(* IEC 61131-3 sources: std_i2980_v2.06_cp053/Source/IMM/ieccontrol/ServiceNet (part 3) *)

         aScan(Execute := FALSE);
      END_IF;
      // next symbol ...
      aScan(Execute := TRUE);
   UNTIL ((NOT aScan.Done) OR (iCntTimeOut = 0))
   END_REPEAT;
ELSE
   // execute false ... clear var outputs and local variables
   bExecuteOld := Execute;
   IF (mHdlNumDataTable <> EMPTY) THEN
      s := KMEM_HashMapL_Delete(mHdlNumDataTable);
      mHdlNumDataTable := EMPTY;
   END_IF;

   iState := 0;
   Error := FALSE;
   sErrMsg := '';
   sParent := '';
   iKeyPosStackIdx := 0;
   ObjRcvCnt := 0;
   iCntStartToken := 0;
   iArrayRecCnt := 0;
   ElapsedTimeSinceLastObj := T#0ms;
END_IF;

@END_Body

@@@BEG_Comment@@@
@TL(39)
@h    ! WARNING !
@h    The Kemro K2 system (including software) only meets category B according to EN 954-1,
@h    thus it is not intended for usage in safety-relevant control applications in the field
@h    of personal safety (e.g. emergency stop).
@h    To implement potentially necessary safety-relevant control tasks, always use additional
@h    external safety devices that are intended for the particular purpose, and meet the necessary
@h    functional safety.
@h    For further information see EN 954-1 (EN ISO 13849-1) and/or the K2-x00 user manual, chapter
@h    "CE conformity, directives and standards".

Algorithm for parsing data stream sent by ServiceNet Server
data presentation: JSON (see http://www.json.org/)

syntax restrictions:
  -> no syntax evaluation of data type "array", tokens within an array are skipped
  -> recursion level for data type "object" is 255 maximum

semantic actions implemented for key - value pairs with values of type "number",
  "true", "false" and "object"

output of parsed data is stored in a hashtable.

objects defined recursive are represented "flat" in same hashtable by adding the parent key
separated by a "." as a prefix to the object key.

the hashtable and it's content is deleted only when reseting input "Execute",
so received data is available in hashtable even if it has not been sent in the
latest message.

data types in hashtable:
-> int numbers, true, false: 4 bytes signed integer (DINT)
-> numbers containing '.' or 'e'/'E': 4 byte float (REAL)

functions available to get a DINT or a REAL value from hashtable.

additionally the parser measures the time since last complete object has
been received for easy timeout detection in calling block.

see documentation for a detailed description.
@@@END_Comment@@@

@BEG_Body
@TL(8)
(**************************************** WARNING ********************************************
 *** The KEBA Kemro K2 System including software is not intended for safety control tasks! ***
 ***                       For further information see Comment tab!                        ***
 *********************************************************************************************)

s := KMEM_HashMapGet(mHdlNumDataTable, Key, Value);
fGetNumValue := s = KMEM_Status_OK;

@END_Body

@@@BEG_Comment@@@
@TL(14)
@h    ! WARNING !
@h    The Kemro K2 system (including software) only meets category B according to EN 954-1,
@h    thus it is not intended for usage in safety-relevant control applications in the field
@h    of personal safety (e.g. emergency stop).
@h    To implement potentially necessary safety-relevant control tasks, always use additional
@h    external safety devices that are intended for the particular purpose, and meet the necessary
@h    functional safety.
@h    For further information see EN 954-1 (EN ISO 13849-1) and/or the K2-x00 user manual, chapter
@h    "CE conformity, directives and standards".

PRIVATE. Not intended to be called from outside this block.

returns the value of a numeric data item stored in hashtable mapped by a certain key
TRUE if found, FALSE in case of an error
@@@END_Comment@@@

@BEG_Body
@TL(15)
(**************************************** WARNING ********************************************
 *** The KEBA Kemro K2 System including software is not intended for safety control tasks! ***
 ***                       For further information see Comment tab!                        ***
 *********************************************************************************************)

bFound := fGetNumValue(Key, tmpValue);
IF ((bFound) AND (tmpValue.dataType = nDTInt)) THEN
   bFound := TRUE;
   ioValue := DWORD_TO_DINT(tmpValue.data);
ELSE
   bFound := FALSE;
END_IF;

fGetDINTValue := bFound;

@END_Body

@@@BEG_Comment@@@
@TL(14)
@h    ! WARNING !
@h    The Kemro K2 system (including software) only meets category B according to EN 954-1,
@h    thus it is not intended for usage in safety-relevant control applications in the field
@h    of personal safety (e.g. emergency stop).
@h    To implement potentially necessary safety-relevant control tasks, always use additional
@h    external safety devices that are intended for the particular purpose, and meet the necessary
@h    functional safety.
@h    For further information see EN 954-1 (EN ISO 13849-1) and/or the K2-x00 user manual, chapter
@h    "CE conformity, directives and standards".

PRIVATE. Not intended to be called from outside this block.

returns the value of a DINT data item stored in hashtable mapped by a certain key
TRUE if found, FALSE in case of an error
@@@END_Comment@@@

@BEG_Body
@TL(18)
(**************************************** WARNING ********************************************
 *** The KEBA Kemro K2 System including software is not intended for safety control tasks! ***
 ***                       For further information see Comment tab!                        ***
 *********************************************************************************************)

IF ((Execute = TRUE) AND (bExecOld = FALSE)) THEN
    // raising edge .. immediate, otherwise if new object recieved since last call
   iCntOld := aParse.ObjRcvCnt - 1;
   bFound := FALSE;
END_IF;

IF (aParse.ObjRcvCnt <> iCntOld) THEN
   bFound := fGetDINTValue(Key, iValue);
   iCntOld := aParse.ObjRcvCnt;
END_IF;

bExecOld := Execute;

@END_Body

@@@BEG_Comment@@@
@TL(15)
@h    ! WARNING !
@h    The Kemro K2 system (including software) only meets category B according to EN 954-1,
@h    thus it is not intended for usage in safety-relevant control applications in the field
@h    of personal safety (e.g. emergency stop).
@h    To implement potentially necessary safety-relevant control tasks, always use additional
@h    external safety devices that are intended for the particular purpose, and meet the necessary
@h    functional safety.
@h    For further information see EN 954-1 (EN ISO 13849-1) and/or the K2-x00 user manual, chapter
@h    "CE conformity, directives and standards".

PRIVATE. Not intended to be called from outside this block.

returns the value of a DINT data item stored in hashtable mapped by a certain key
if not found on raising edge of Execute,
the algorithm will try to find the value each time a new object has been parsed
@@@END_Comment@@@

@BEG_Body
@TL(11)
(**************************************** WARNING ********************************************
 *** The KEBA Kemro K2 System including software is not intended for safety control tasks! ***
 ***                       For further information see Comment tab!                        ***
 *********************************************************************************************)

bFound := fGetNumValue(Key, tmpValue);
IF (bFound) THEN
   bFound := CONVERT_DWORD_TO_REAL(tmpValue.data, rValue);
END_IF;
fGetRealValue := bFound;

@END_Body

@@@BEG_Comment@@@
@TL(14)
@h    ! WARNING !
@h    The Kemro K2 system (including software) only meets category B according to EN 954-1,
@h    thus it is not intended for usage in safety-relevant control applications in the field
@h    of personal safety (e.g. emergency stop).
@h    To implement potentially necessary safety-relevant control tasks, always use additional
@h    external safety devices that are intended for the particular purpose, and meet the necessary
@h    functional safety.
@h    For further information see EN 954-1 (EN ISO 13849-1) and/or the K2-x00 user manual, chapter
@h    "CE conformity, directives and standards".

PRIVATE. Not intended to be called from outside this block.

returns the value of a REAL data item stored in hashtable mapped by a certain key
TRUE if found, FALSE in case of an error
@@@END_Comment@@@

@BEG_Body
@TL(18)
(**************************************** WARNING ********************************************
 *** The KEBA Kemro K2 System including software is not intended for safety control tasks! ***
 ***                       For further information see Comment tab!                        ***
 *********************************************************************************************)

IF ((Execute = TRUE) AND (bExecOld = FALSE)) THEN
   // raising edge .. immediate, otherwise if new object recieved since last call
   iCntOld := aParse.ObjRcvCnt - 1;
   bFound := FALSE;
END_IF;

IF (aParse.ObjRcvCnt <> iCntOld) THEN
   bFound := fGetRealValue(Key, rValue);
   iCntOld := aParse.ObjRcvCnt;
END_IF;

bExecOld := Execute;

@END_Body

@@@BEG_Comment@@@
@TL(13)
@h    ! WARNING !
@h    The Kemro K2 system (including software) only meets category B according to EN 954-1,
@h    thus it is not intended for usage in safety-relevant control applications in the field
@h    of personal safety (e.g. emergency stop).
@h    To implement potentially necessary safety-relevant control tasks, always use additional
@h    external safety devices that are intended for the particular purpose, and meet the necessary
@h    functional safety.
@h    For further information see EN 954-1 (EN ISO 13849-1) and/or the K2-x00 user manual, chapter
@h    "CE conformity, directives and standards".

returns the value of a REAL data item stored in hashtable mapped by a certain key
if not found on raising edge of Execute,
the algorithm will try to find the value each time a new object has been parsed
@@@END_Comment@@@
@END_Body

@END_Contents

(* ---- ABRemoteMaintenance.pu ---- *)
(*
@h    ! WARNING !
@h    The Kemro K2 system (including software) only meets category B according to EN 954-1,
@h    thus it is not intended for usage in safety-relevant control applications in the field
@h    of personal safety (e.g. emergency stop).
@h    To implement potentially necessary safety-relevant control tasks, always use additional
@h    external safety devices that are intended for the particular purpose, and meet the necessary
@h    functional safety.
@h    For further information see EN 954-1 (EN ISO 13849-1) and/or the K2-x00 user manual, chapter
@h    "CE conformity, directives and standards".

This AB controls the logic for connecting ServiceNet via the ServiceNet embedded functionality
via the Remote Maintenance software unit.
*)

IMPORT_OVER_LISTFILE
 KSYS_BPAPI_VAR_READ
, KSYS_BPAPI_VAR_WRITE
, GET_RUNTIME
, KCAT_GetValue
, KCAT_GetHandle
, STOP_PROCESS_ALGORITHM
, START_PROCESS_ALGORITHM
, TOLOWER
, cKSYS_BPApiStateOk
, tsNetworkCfg
, tsTraceLevel
, tsSiteManagerStatus
, TON
, KSYS_BPApiState
, KCAT_HandleData
, KCAT_Status

END_IMPORT

ALGORITHM_BLOCK ABRemoteMaintenance #DUMMY_EDIT_BLOCK

SYSTEM_VAR
 sv_SNNetworkConfig : tsNetworkCfg (* network config to use when connecting to servicenet *);
 sv_iCpuId : LINT;
 sv_TraceLevel : tsTraceLevel;
 sv_bRemoteMaintAvailable : BOOL (* True, if the remote maintenance service is available (Linux only) *);
 sv_bRemoteMaintActivate : BOOL (* Set to true, to activate the remote maintenance *);
 sv_bRemoteMaintActivated : BOOL (* True, if the remote maintenance is activated *);
 sv_sSiteManagerSetServer : STRING(255) (* The SiteManager server name to connect *);
 sv_sSiteManagerSetName : STRING(255) (* The SiteManager domain to connect *);
 sv_iRemoteMaintState : UDINT (* State of the remote maintenance service (1=active) *);
 sv_SiteManager : tsSiteManagerStatus (* Secomea SiteManager structure *);
 sv_bInitStart : BOOL;
END_VAR

SYSTEM_OBJECT
 TaskVis : TASK;
 TaskVisLow : TASK;
END_OBJECT

VAR
 fbTimer : TON;
 mbInit : BOOL;
END_VAR

ALGORITHM aReadSiteManagerStatus

VAR
 SysState : KSYS_BPApiState;
 sTmp : STRING(255);
 dummy : DINT;
END_VAR
#BEGIN_EDIT_BLOCK
(**************************************** WARNING ********************************************
 *** The KEBA Kemro K2 System including software is not intended for safety control tasks! ***
 ***                       For further information see Comment tab!                        ***
 *********************************************************************************************)

SysState := KSYS_BPAPI_VAR_READ('SYS.SERVICES.RemoteMaintenance.Secomea.Sitemanager.status', sTmp);
IF(SysState = cKSYS_BPApiStateOk) THEN
   sv_SiteManager.sState := sTmp;
ELSIF(sv_TraceLevel.bApplication) THEN
   dummy := Print("Remote maintenance: Site manager status cant be read");
END_IF;

SysState := KSYS_BPAPI_VAR_TXTREAD('SYS.SERVICES.RemoteMaintenance.Secomea.Sitemanager.color', sTmp);
IF(SysState = cKSYS_BPApiStateOk) THEN
   sTmp := TOLOWER(sTmp);
   sv_SiteManager.sColor := sTmp;

   // currently the modem status can only be determined with the status string returned
   IF(sTmp = 'red') THEN
      sv_SiteManager.iState := 1;
   ELSIF(sTmp = 'yellow') THEN
      sv_SiteManager.iState := 2;
   ELSIF(sTmp = 'green') THEN
      sv_SiteManager.iState := 3;
   ELSIF(sTmp = 'blue') THEN
      sv_SiteManager.iState := 4;
   ELSE
      sv_SiteManager.iState := 0;
   END_IF;

   sv_SiteManager.bConnected := (sv_SiteManager.iState = 4);

ELSIF(sv_TraceLevel.bApplication) THEN
   dummy := Print("Remote maintenance: Site manager color cant be read");
   sv_SiteManager.bConnected := FALSE;
END_IF;

;#END_EDIT_BLOCK END_ALGORITHM

ALGORITHM aReadSiteManagerServer

VAR
 SysState : KSYS_BPApiState;
 sTmp : STRING(255);
 dummy : DINT;
END_VAR
#BEGIN_EDIT_BLOCK
(**************************************** WARNING ********************************************
 *** The KEBA Kemro K2 System including software is not intended for safety control tasks! ***
 ***                       For further information see Comment tab!                        ***
 *********************************************************************************************)

SysState := KSYS_BPAPI_VAR_TXTREAD('SYS.CFG.Secomea.Sitemanager.Server', sTmp);
IF(SysState = cKSYS_BPApiStateOk) THEN
   sv_SiteManager.sServer := sTmp;
ELSIF(sv_TraceLevel.bApplication) THEN
   dummy := Print("Remote maintenance: Site manager server cant be read");
END_IF;

SysState := KSYS_BPAPI_VAR_TXTREAD('SYS.CFG.Secomea.Sitemanager.Name', sTmp);
IF(SysState = cKSYS_BPApiStateOk) THEN
   sv_SiteManager.sName := sTmp;
ELSIF(sv_TraceLevel.bApplication) THEN
   dummy := Print("Remote maintenance: Site manager name cant be read");
END_IF;

SysState := KSYS_BPAPI_VAR_TXTREAD('SYS.CFG.Secomea.Sitemanager.Domain', sTmp);
IF(SysState = cKSYS_BPApiStateOk) THEN
   sv_SiteManager.sDomain := sTmp;
ELSIF(sv_TraceLevel.bApplication) THEN
   dummy := Print("Remote maintenance: Site manager domain cant be read");
END_IF;

;#END_EDIT_BLOCK END_ALGORITHM

PROCESS_ALGORITHM paRun ON TaskVisLow

VAR
 iRemoteMaintState : UDINT;
 SysState : KSYS_BPApiState;
 dummy : DINT;
 t : TIME;
 iTime : DINT;
 iStep : DINT;
END_VAR
#BEGIN_EDIT_BLOCK
(**************************************** WARNING ********************************************
 *** The KEBA Kemro K2 System including software is not intended for safety control tasks! ***
 ***                       For further information see Comment tab!                        ***
 *********************************************************************************************)

t := GET_RUNTIME();

IF iStep = 0 THEN
   fbTimer(IN := FALSE, PT := t#500ms);
   iStep := 1;
END_IF;

IF iStep = 1 THEN
   fbTimer(IN := TRUE);
   IF(fbTimer.Q) THEN
      iStep := 5;
   END_IF;
END_IF;

IF iStep = 5 THEN
   SysState := KSYS_BPAPI_VAR_READ('SYS.SERVICES.RemoteMaintenance.Secomea.state', iRemoteMaintState);
   IF(SysState <> cKSYS_BPApiStateOk) THEN
      IF(sv_TraceLevel.bApplication) THEN
         dummy := Print("Remote maintenance service not found, KSYS_BPApiState %x", SysState);
      END_IF;
      sv_bRemoteMaintAvailable := FALSE;
      STOP_PROCESS_ALGORITHM(paRun);
      RETURN;
   END_IF;

   IF iRemoteMaintState <> 0 THEN
      // continuously poll for the connection status if the state is active
      // IEC does not have a method for post-updating a BPAPI variable
      aReadSiteManagerStatus();
   ELSIF sv_iRemoteMaintState <> 0 THEN
      // reset the connection status
      IF(sv_SiteManager.sState <> 'disabled') THEN
         sv_SiteManager.sState := 'disabled';
      END_IF;
      IF(sv_SiteManager.sColor <> '') THEN
         sv_SiteManager.sColor := '';
         sv_SiteManager.iState := 0;
      END_IF;
      sv_SiteManager.bConnected := FALSE;
   END_IF;

   sv_iRemoteMaintState := iRemoteMaintState;

   fbTimer(IN := FALSE);
   iStep := 0;
END_IF;

t := GET_RUNTIME() - t;
iTime := LINT_TO_DINT(TIME_TO_LINT(t) / 1000);
IF(iTime >= 10 AND sv_TraceLevel.bApplication) THEN
   dummy := Print("Remote maintenance: Runtime of ABRemoteMaintenance.paRun %d ms", iTime);
END_IF;

;#END_EDIT_BLOCK END_ALGORITHM

POSTUPDATE_ALGORITHM pUpdateServer ON TaskVis WITH sv_sSiteManagerSetServer

VAR
 dummy : DINT;
 SysState : KSYS_BPApiState;
END_VAR
#BEGIN_EDIT_BLOCK
(**************************************** WARNING ********************************************
 *** The KEBA Kemro K2 System including software is not intended for safety control tasks! ***
 ***                       For further information see Comment tab!                        ***
 *********************************************************************************************)

IF (NOT mbInit) THEN
   RETURN;
END_IF;

IF(sv_bRemoteMaintAvailable) THEN
   SysState := KSYS_BPAPI_VAR_WRITE('SYS.CFG.Secomea.Sitemanager.Server', sv_sSiteManagerSetServer);
   IF(SysState <> cKSYS_BPApiStateOk) THEN
      dummy := Print("Remote maintenance: Could not set site manager server, KSYS_BPApiState %x", SysState);
      sv_bRemoteMaintActivate := FALSE;
   END_IF;

   aReadSiteManagerServer();

END_IF;

;#END_EDIT_BLOCK END_ALGORITHM

POSTUPDATE_ALGORITHM pUpdateName ON TaskVis WITH sv_sSiteManagerSetName

VAR
 dummy : DINT;
 SysState : KSYS_BPApiState;
 sTmp : STRING(255);
END_VAR
#BEGIN_EDIT_BLOCK
(**************************************** WARNING ********************************************
 *** The KEBA Kemro K2 System including software is not intended for safety control tasks! ***
 ***                       For further information see Comment tab!                        ***
 *********************************************************************************************)

IF (NOT mbInit) THEN
   RETURN;
END_IF;

IF(sv_bRemoteMaintAvailable) THEN

   sTmp := CONCAT(LINT_TO_STRING(sv_iCpuId), '_', sv_sSiteManagerSetName);
   SysState := KSYS_BPAPI_VAR_WRITE('SYS.CFG.Secomea.Sitemanager.Name', sTmp);
   IF(SysState <> cKSYS_BPApiStateOk) THEN
      dummy := Print("Remote maintenance: Could not set site manager name, KSYS_BPApiState %x", SysState);
      sv_bRemoteMaintActivate := FALSE;
   END_IF;

   aReadSiteManagerServer();

END_IF;

;#END_EDIT_BLOCK END_ALGORITHM

POSTUPDATE_ALGORITHM pInit ON TaskVis WITH sv_bInitStart

VAR
 dummy : DINT;
 SysState : KSYS_BPApiState;
 iRemoteMaintState : UDINT;
 bRemoteMaintActive : BOOL;
 sSecomeaDomain : STRING(255);
 iTemp : DINT;
 b : BOOL;
 bLinux : BOOL;
 HandleData : KCAT_HandleData;
 Status : KCAT_Status;
 sTemp : STRING(255);
 sFind : STRING(32);
END_VAR
#BEGIN_EDIT_BLOCK
(**************************************** WARNING ********************************************
 *** The KEBA Kemro K2 System including software is not intended for safety control tasks! ***
 ***                       For further information see Comment tab!                        ***
 *********************************************************************************************)

HandleData := KCAT_GetHandle('UOS.System');
IF HandleData.Status = KCAT_Status_OK THEN
   Status := KCAT_GetValue(Handle := HandleData.Handle, Buffer := sTemp);
   IF (sTemp = 'Linux') THEN
      bLinux := TRUE;
   END_IF;
END_IF;

IF(NOT bLinux) THEN
   // do not create the nodes on VxWorks - this info does not exist
   // stop and return
   sv_bRemoteMaintAvailable := FALSE;
   STOP_PROCESS_ALGORITHM(paRun);
   RETURN;
END_IF;

// check if RemoteMaintenance software unit is present
SysState := KSYS_BPAPI_VAR_READ('SYS.SERVICES.RemoteMaintenance.Secomea.state', iRemoteMaintState);
IF(SysState <> cKSYS_BPApiStateOk) THEN
   IF(sv_TraceLevel.bApplication) THEN
      dummy := Print("Remote maintenance: service/state not found - stopping, KSYS_BPApiState %x", SysState);
   END_IF;
   // stop and return
   sv_bRemoteMaintAvailable := FALSE;
   STOP_PROCESS_ALGORITHM(paRun);
   RETURN;
END_IF;

// Domain must also be configured
SysState := KSYS_BPAPI_VAR_READ('SYS.CFG.Secomea.Sitemanager.Domain', sSecomeaDomain);
IF(SysState <> cKSYS_BPApiStateOk) THEN
   IF(sv_TraceLevel.bApplication) THEN
      dummy := Print("Remote maintenance: service/domain not found - stopping, KSYS_BPApiState %x", SysState);
   END_IF;
   // stop and return
   sv_bRemoteMaintAvailable := FALSE;
   STOP_PROCESS_ALGORITHM(paRun);
   RETURN;
END_IF;

SysState := KSYS_BPAPI_VAR_READ('SYS.SERVICES.RemoteMaintenance.Secomea.activated', bRemoteMaintActive);
IF(SysState <> cKSYS_BPApiStateOk) THEN
   dummy := Print("Remote maintenance: activated flag not found - setting ignored, KSYS_BPApiState %x", SysState);
   RETURN;
END_IF;
sv_bRemoteMaintActivated := bRemoteMaintActive;
b := WRITE_SV_DIRECT(sv_bRemoteMaintActivate, bRemoteMaintActive);

aReadSiteManagerStatus();
aReadSiteManagerServer();

// initialize the setter variables
sv_sSiteManagerSetServer := sv_SiteManager.sServer;

// prepend <CPUID>_ to the display string
sFind := CONCAT(LINT_TO_STRING(sv_iCpuId), '_');
iTemp := FIND(sv_SiteManager.sName, sFind);

IF (iTemp = 1) THEN
   sv_sSiteManagerSetName := RIGHT(sv_SiteManager.sName, LEN(sv_SiteManager.sName)- LEN(sFind));
ELSE
   sv_sSiteManagerSetName := sv_SiteManager.sName;
END_IF;

sv_iRemoteMaintState := iRemoteMaintState;

// disable ServiceNet IP-switching per default
sv_SNNetworkConfig.sIP := '';

// RemoteMaintenance is available start polling for status changes
sv_bRemoteMaintAvailable := TRUE;
START_PROCESS_ALGORITHM(paRun);

mbInit := TRUE;

;#END_EDIT_BLOCK END_ALGORITHM

POSTUPDATE_ALGORITHM pActivate ON TaskVis WITH sv_bRemoteMaintActivate

VAR
 bRemoteMaintActive : BOOL;
 SysState : KSYS_BPApiState;
 dummy : DINT;
END_VAR
#BEGIN_EDIT_BLOCK
(**************************************** WARNING ********************************************
 *** The KEBA Kemro K2 System including software is not intended for safety control tasks! ***
 ***                       For further information see Comment tab!                        ***
 *********************************************************************************************)

// read the current activation status
SysState := KSYS_BPAPI_VAR_READ('SYS.SERVICES.RemoteMaintenance.Secomea.activated', bRemoteMaintActive);
IF(SysState <> cKSYS_BPApiStateOk) THEN
   dummy := Print("Remote maintenance: activated flag not found - setting ignored, KSYS_BPApiState %x", SysState);
   RETURN;
END_IF;

IF(sv_bRemoteMaintActivate = bRemoteMaintActive) THEN
   sv_bRemoteMaintActivated := bRemoteMaintActive;
   RETURN;
END_IF;

// activate service
SysState := KSYS_BPAPI_VAR_WRITE('SYS.SERVICES.RemoteMaintenance.Secomea.activated', sv_bRemoteMaintActivate);
IF(SysState <> cKSYS_BPApiStateOk) THEN
   dummy := Print("Remote maintenance: activated flag not found - could not set, KSYS_BPApiState %x", SysState);
   sv_bRemoteMaintActivate := FALSE;
   RETURN;
END_IF;

sv_bRemoteMaintActivated := sv_bRemoteMaintActivate;

;#END_EDIT_BLOCK END_ALGORITHM

END_ALGORITHM_BLOCK

#END_OF_IEC_PART

@Puma @IecEditor 6 180 @Pou 25
@@@BEG_Comment@@@
@h    ! WARNING !
@h    The Kemro K2 system (including software) only meets category B according to EN 954-1,
@h    thus it is not intended for usage in safety-relevant control applications in the field
@h    of personal safety (e.g. emergency stop).
@h    To implement potentially necessary safety-relevant control tasks, always use additional
@h    external safety devices that are intended for the particular purpose, and meet the necessary
@h    functional safety.
@h    For further information see EN 954-1 (EN ISO 13849-1) and/or the K2-x00 user manual, chapter
@h    "CE conformity, directives and standards".

This AB controls the logic for connecting ServiceNet via the ServiceNet embedded functionality
via the Remote Maintenance software unit.
@@@END_Comment@@@

@BEG_Contents

@BEG_Func
@RT(17)FuncTreeContainer
8
@Var @RT(19)KSYS_BPAPI_VAR_READ @RT(0) @T @T @DERIVED 0 @F @RT(22)KEBA_STANDARD_FUNCTION @F
@T
@BEG_Attrib
0 @RT(0) @RT(0)
@END_Attrib
1 1 @F @F @F @F

@Var @RT(20)KSYS_BPAPI_VAR_WRITE @RT(0) @T @T @DERIVED 0 @F @RT(22)KEBA_STANDARD_FUNCTION @F
@T
@BEG_Attrib
0 @RT(0) @RT(0)
@END_Attrib
1 1 @F @F @F @F

@Var @RT(11)GET_RUNTIME @RT(0) @T @T @DERIVED 0 @F @RT(22)KEBA_STANDARD_FUNCTION @F
@T
@BEG_Attrib
0 @RT(0) @RT(0)
@END_Attrib
1 1 @F @F @F @F

@Var @RT(13)KCAT_GetValue @RT(0) @T @T @DERIVED 0 @F @RT(22)KEBA_STANDARD_FUNCTION @F
@T
@BEG_Attrib
0 @RT(0) @RT(0)
@END_Attrib
1 1 @F @F @F @F

@Var @RT(14)KCAT_GetHandle @RT(0) @T @T @DERIVED 0 @F @RT(22)KEBA_STANDARD_FUNCTION @F
@T
@BEG_Attrib
0 @RT(0) @RT(0)
@END_Attrib
1 1 @F @F @F @F

@Var @RT(22)STOP_PROCESS_ALGORITHM @RT(0) @T @T @DERIVED 0 @F @RT(23)KEBA_STANDARD_PROCEDURE @F
@T
@BEG_Attrib
0 @RT(0) @RT(0)
@END_Attrib
1 1 @F @F @F @F

@Var @RT(23)START_PROCESS_ALGORITHM @RT(0) @T @T @DERIVED 0 @F @RT(23)KEBA_STANDARD_PROCEDURE @F
@T
@BEG_Attrib
0 @RT(0) @RT(0)
@END_Attrib
1 1 @F @F @F @F

@Var @RT(7)TOLOWER @RT(0) @T @T @DERIVED 0 @F @RT(22)KEBA_STANDARD_FUNCTION @F
@T
@BEG_Attrib
0 @RT(0) @RT(0)
@END_Attrib
1 1 @F @F @F @F

@END_Func

@BEG_Const
@RT(18)ConstTreeContainer
1
@Var @RT(18)cKSYS_BPApiStateOk @RT(0) @T @F @DT @RT(5)DWORD @RT(0) @T @T @BASIC 0 @F
@F @F
@T
@BEG_Attrib
0 @RT(4)16#0 @RT(0)
@END_Attrib
1 1 @F @F @F @F

@END_Const

@BEG_Export

@BEG_Kind
@ALGORITHM_BLOCK @RT(19)ABRemoteMaintenance @STRUCTURED_TEXT
@RT(0) @RT(0) @RT(0)
@END_Kind

@BEG_Dcl
@RT(16)DclTreeContainer
15
@Var @RT(7)TaskVis @RT(0) @T @T @RENAMED 0 @T @T @DT @RT(4)TASK @RT(0) @T @T @BASIC 0 @F
@F @F
@T
@BEG_Attrib
3 @RT(0) @RT(0) @RT(0)
@END_Attrib
1 7 @F @F @F @F

@Var @RT(10)TaskVisLow @RT(0) @T @T @RENAMED 0 @T @T @DT @RT(4)TASK @RT(0) @T @T @BASIC 0 @F
@F @F
@T
@BEG_Attrib
3 @RT(0) @RT(0) @RT(0)
@END_Attrib
1 7 @F @F @F @F

@Var @RT(18)sv_SNNetworkConfig @RT(0) @T @T @DERIVED 0 @T @T @DT @RT(12)tsNetworkCfg @RT(0) @T @T @UNKNOWN 0 @F
@F @F
@T
@BEG_Attrib
3 @RT(0) @RT(51)network config to use when connecting to servicenet @RT(0)
@END_Attrib
1 8 @F @F @F @F

@Var @RT(9)sv_iCpuId @RT(0) @T @F @DT @RT(4)LINT @RT(0) @T @T @BASIC 0 @F
@F @F
@T
@BEG_Attrib
3 @RT(0) @RT(0) @RT(0)
@END_Attrib
1 8 @F @F @F @F

@Var @RT(13)sv_TraceLevel @RT(0) @T @T @DERIVED 0 @T @T @DT @RT(12)tsTraceLevel @RT(0) @T @T @UNKNOWN 0 @F
@F @F
@T
@BEG_Attrib
3 @RT(0) @RT(0) @RT(0)
@END_Attrib
1 8 @F @F @F @F

@Var @RT(24)sv_bRemoteMaintAvailable @RT(0) @T @F @DT @RT(4)BOOL @RT(0) @T @T @BASIC 0 @F
@F @F
@T
@BEG_Attrib
3 @RT(0) @RT(65)True, if the remote maintenance service is available (Linux only) @RT(0)
@END_Attrib
1 8 @F @F @F @F

@Var @RT(23)sv_bRemoteMaintActivate @RT(0) @T @T @RENAMED 0 @T @T @DT @RT(4)BOOL @RT(0) @T @T @BASIC 0 @F
@F @F
@T
@BEG_Attrib
3 @RT(0) @RT(47)Set to true, to activate the remote maintenance @RT(0)
@END_Attrib
1 8 @F @F @F @F

@Var @RT(24)sv_bRemoteMaintActivated @RT(0) @T @F @DT @RT(4)BOOL @RT(0) @T @T @BASIC 0 @F
@F @F
@T
@BEG_Attrib
3 @RT(0) @RT(44)True, if the remote maintenance is activated @RT(0)
@END_Attrib
1 8 @F @F @F @F

@Var @RT(24)sv_sSiteManagerSetServer @RT(0) @T @F @DT @RT(11)STRING(255) @RT(0) @T @T @STRING 0 @F @RT(3)255 @F
@F @F
@T
@BEG_Attrib
3 @RT(0) @RT(38)The SiteManager server name to connect @RT(0)
@END_Attrib
1 8 @F @F @F @F

@Var @RT(22)sv_sSiteManagerSetName @RT(0) @T @F @DT @RT(11)STRING(255) @RT(0) @T @T @STRING 0 @F @RT(3)255 @F
@F @F
@T
@BEG_Attrib
3 @RT(0) @RT(33)The SiteManager domain to connect @RT(0)
@END_Attrib
1 8 @F @F @F @F

@Var @RT(20)sv_iRemoteMaintState @RT(0) @T @F @DT @RT(5)UDINT @RT(0) @T @T @BASIC 0 @F
@F @F
@T
@BEG_Attrib
3 @RT(0) @RT(50)State of the remote maintenance service (1=active) @RT(0)
@END_Attrib
1 8 @F @F @F @F

@Var @RT(14)sv_SiteManager @RT(0) @T @T @DERIVED 0 @T @T @DT @RT(19)tsSiteManagerStatus @RT(0) @T @T @UNKNOWN 0 @F
@F @F
@T
@BEG_Attrib
3 @RT(0) @RT(29)Secomea SiteManager structure @RT(0)
@END_Attrib
1 8 @F @F @F @F

@Var @RT(7)fbTimer @RT(0) @T @T @DERIVED 0 @T @T @DT @RT(3)TON @RT(0) @T @T @UNKNOWN 0 @F
@F @F
@T
@BEG_Attrib
3 @RT(0) @RT(0) @RT(0)
@END_Attrib
1 0 @F @F @F @F

@Var @RT(6)mbInit @RT(0) @T @F @DT @RT(4)BOOL @RT(0) @T @T @BASIC 0 @F
@F @F
@T
@BEG_Attrib
3 @RT(0) @RT(0) @RT(0)
@END_Attrib
1 0 @F @F @F @F

@Var @RT(13)sv_bInitStart @RT(0) @T @T @RENAMED 0 @T @T @DT @RT(4)BOOL @RT(0) @T @T @BASIC 0 @F
@F @F
@T
@BEG_Attrib
3 @RT(0) @RT(0) @RT(0)
@END_Attrib
1 8 @F @F @F @F

@END_Dcl

@END_Export

@BEG_Body

7

@BEG_Export

@BEG_Algo
@ALGORITHM @RT(22)aReadSiteManagerStatus @STRUCTURED_TEXT
@RT(0) @RT(0) @RT(0) @F @F
@END_Algo

@BEG_Dcl
@RT(16)DclTreeContainer
3
@Var @RT(8)SysState @RT(0) @T @T @DERIVED 0 @T @T @DT @RT(15)KSYS_BPApiState @RT(0) @T @T @UNKNOWN 0 @F
@F @F
@T
@BEG_Attrib
3 @RT(0) @RT(0) @RT(0)
@END_Attrib
1 0 @F @F @F @F

@Var @RT(4)sTmp @RT(0) @T @F @DT @RT(11)STRING(255) @RT(0) @T @T @STRING 0 @F @RT(3)255 @F
@F @F
@T
@BEG_Attrib
3 @RT(0) @RT(0) @RT(0)
@END_Attrib
1 0 @F @F @F @F

@Var @RT(5)dummy @RT(0) @T @F @DT @RT(4)DINT @RT(0) @T @T @BASIC 0 @F
@F @F
@T
@BEG_Attrib
3 @RT(0) @RT(0) @RT(0)
@END_Attrib
1 0 @F @F @F @F

@END_Dcl

@END_Export

@BEG_Export

@BEG_Algo
@ALGORITHM @RT(22)aReadSiteManagerServer @STRUCTURED_TEXT
@RT(0) @RT(0) @RT(0) @F @F
@END_Algo

@BEG_Dcl
@RT(16)DclTreeContainer
3
@Var @RT(8)SysState @RT(0) @T @T @DERIVED 0 @T @T @DT @RT(15)KSYS_BPApiState @RT(0) @T @T @UNKNOWN 0 @F
@F @F
@T
@BEG_Attrib
3 @RT(0) @RT(0) @RT(0)
@END_Attrib
1 0 @F @F @F @F

@Var @RT(4)sTmp @RT(0) @T @F @DT @RT(11)STRING(255) @RT(0) @T @T @STRING 0 @F @RT(3)255 @F
@F @F
@T
@BEG_Attrib
3 @RT(0) @RT(0) @RT(0)
@END_Attrib
1 0 @F @F @F @F

@Var @RT(5)dummy @RT(0) @T @F @DT @RT(4)DINT @RT(0) @T @T @BASIC 0 @F
@F @F
@T
@BEG_Attrib
3 @RT(0) @RT(0) @RT(0)
@END_Attrib
1 0 @F @F @F @F

@END_Dcl

@END_Export

@BEG_Export

@BEG_Algo
@PROCESS_ALGORITHM @RT(5)paRun @STRUCTURED_TEXT
@RT(0) @RT(0) @RT(10)TaskVisLow @F @F
@END_Algo

@BEG_Dcl
@RT(16)DclTreeContainer
6
@Var @RT(17)iRemoteMaintState @RT(0) @T @F @DT @RT(5)UDINT @RT(0) @T @T @BASIC 0 @F
@F @F
@T
@BEG_Attrib
3 @RT(0) @RT(0) @RT(0)
@END_Attrib
1 0 @F @F @F @F

@Var @RT(8)SysState @RT(0) @T @T @DERIVED 0 @T @T @DT @RT(15)KSYS_BPApiState @RT(0) @T @T @UNKNOWN 0 @F
@F @F
@T
@BEG_Attrib
3 @RT(0) @RT(0) @RT(0)
@END_Attrib
1 0 @F @F @F @F

@Var @RT(5)dummy @RT(0) @T @F @DT @RT(4)DINT @RT(0) @T @T @BASIC 0 @F
@F @F
@T
@BEG_Attrib
3 @RT(0) @RT(0) @RT(0)
@END_Attrib
1 0 @F @F @F @F

@Var @RT(1)t @RT(0) @T @F @DT @RT(4)TIME @RT(0) @T @T @BASIC 0 @F
@F @F
@T
@BEG_Attrib
3 @RT(0) @RT(0) @RT(0)
@END_Attrib
1 0 @F @F @F @F

@Var @RT(5)iTime @RT(0) @T @F @DT @RT(4)DINT @RT(0) @T @T @BASIC 0 @F
@F @F
@T
@BEG_Attrib
3 @RT(0) @RT(0) @RT(0)
@END_Attrib
1 0 @F @F @F @F

@Var @RT(5)iStep @RT(0) @T @F @DT @RT(4)DINT @RT(0) @T @T @BASIC 0 @F
@F @F
@T
@BEG_Attrib
3 @RT(0) @RT(0) @RT(0)
@END_Attrib
1 0 @F @F @F @F

@END_Dcl

@END_Export

@BEG_Export

@BEG_Algo
@POSTUPDATE_ALGORITHM @RT(13)pUpdateServer @STRUCTURED_TEXT
@RT(0) @RT(24)sv_sSiteManagerSetServer @RT(7)TaskVis @F @F
@END_Algo

@BEG_Dcl
@RT(16)DclTreeContainer
2
@Var @RT(5)dummy @RT(0) @T @F @DT @RT(4)DINT @RT(0) @T @T @BASIC 0 @F
@F @F
@T
@BEG_Attrib
3 @RT(0) @RT(0) @RT(0)
@END_Attrib
1 0 @F @F @F @F

@Var @RT(8)SysState @RT(0) @T @T @DERIVED 0 @T @T @DT @RT(15)KSYS_BPApiState @RT(0) @T @T @UNKNOWN 0 @F
@F @F
@T
@BEG_Attrib
3 @RT(0) @RT(0) @RT(0)
@END_Attrib
1 0 @F @F @F @F

@END_Dcl

@END_Export

@BEG_Export

@BEG_Algo
@POSTUPDATE_ALGORITHM @RT(11)pUpdateName @STRUCTURED_TEXT
@RT(0) @RT(22)sv_sSiteManagerSetName @RT(7)TaskVis @F @F
@END_Algo

@BEG_Dcl
@RT(16)DclTreeContainer
3
@Var @RT(5)dummy @RT(0) @T @F @DT @RT(4)DINT @RT(0) @T @T @BASIC 0 @F
@F @F
@T
@BEG_Attrib
3 @RT(0) @RT(0) @RT(0)
@END_Attrib
1 0 @F @F @F @F

@Var @RT(8)SysState @RT(0) @T @T @DERIVED 0 @T @T @DT @RT(15)KSYS_BPApiState @RT(0) @T @T @UNKNOWN 0 @F
@F @F
@T
@BEG_Attrib
3 @RT(0) @RT(0) @RT(0)
@END_Attrib
1 0 @F @F @F @F

@Var @RT(4)sTmp @RT(0) @T @F @DT @RT(11)STRING(255) @RT(0) @T @T @STRING 0 @F @RT(3)255 @F
@F @F
@T
@BEG_Attrib
3 @RT(0) @RT(0) @RT(0)
@END_Attrib
1 0 @F @F @F @F

@END_Dcl

@END_Export

@BEG_Export

@BEG_Algo
@POSTUPDATE_ALGORITHM @RT(5)pInit @STRUCTURED_TEXT
@RT(0) @RT(13)sv_bInitStart @RT(7)TaskVis @F @F
@END_Algo

@BEG_Dcl
@RT(16)DclTreeContainer
12
@Var @RT(5)dummy @RT(0) @T @F @DT @RT(4)DINT @RT(0) @T @T @BASIC 0 @F
@F @F
@T
@BEG_Attrib
3 @RT(0) @RT(0) @RT(0)
@END_Attrib
1 0 @F @F @F @F

@Var @RT(8)SysState @RT(0) @T @T @DERIVED 0 @T @T @DT @RT(15)KSYS_BPApiState @RT(0) @T @T @UNKNOWN 0 @F
@F @F
@T
@BEG_Attrib
3 @RT(0) @RT(0) @RT(0)
@END_Attrib
1 0 @F @F @F @F

@Var @RT(17)iRemoteMaintState @RT(0) @T @F @DT @RT(5)UDINT @RT(0) @T @T @BASIC 0 @F
@F @F
@T
@BEG_Attrib
3 @RT(0) @RT(0) @RT(0)
@END_Attrib
1 0 @F @F @F @F

@Var @RT(18)bRemoteMaintActive @RT(0) @T @F @DT @RT(4)BOOL @RT(0) @T @T @BASIC 0 @F
@F @F
@T
@BEG_Attrib
3 @RT(0) @RT(0) @RT(0)
@END_Attrib
1 0 @F @F @F @F

@Var @RT(14)sSecomeaDomain @RT(0) @T @F @DT @RT(11)STRING(255) @RT(0) @T @T @STRING 0 @F @RT(3)255 @F
@F @F
@T
@BEG_Attrib
3 @RT(0) @RT(0) @RT(0)
@END_Attrib
1 0 @F @F @F @F

@Var @RT(5)iTemp @RT(0) @T @F @DT @RT(4)DINT @RT(0) @T @T @BASIC 0 @F
@F @F
@T
@BEG_Attrib
3 @RT(0) @RT(0) @RT(0)
@END_Attrib
1 0 @F @F @F @F

@Var @RT(1)b @RT(0) @T @F @DT @RT(4)BOOL @RT(0) @T @T @BASIC 0 @F
@F @F
@T
@BEG_Attrib
3 @RT(0) @RT(0) @RT(0)
@END_Attrib
1 0 @F @F @F @F

@Var @RT(6)bLinux @RT(0) @T @F @DT @RT(4)BOOL @RT(0) @T @T @BASIC 0 @F
@F @F
@T
@BEG_Attrib
3 @RT(0) @RT(0) @RT(0)
@END_Attrib
1 0 @F @F @F @F

@Var @RT(10)HandleData @RT(0) @T @T @DERIVED 0 @T @T @DT @RT(15)KCAT_HandleData @RT(0) @T @T @UNKNOWN 0 @F
@F @F
@T
@BEG_Attrib
3 @RT(0) @RT(0) @RT(0)
@END_Attrib
1 0 @F @F @F @F

@Var @RT(6)Status @RT(0) @T @T @DERIVED 0 @T @T @DT @RT(11)KCAT_Status @RT(0) @T @T @UNKNOWN 0 @F
@F @F
@T
@BEG_Attrib
3 @RT(0) @RT(0) @RT(0)
@END_Attrib
1 0 @F @F @F @F

@Var @RT(5)sTemp @RT(0) @T @F @DT @RT(11)STRING(255) @RT(0) @T @T @STRING 0 @F @RT(3)255 @F
@F @F
@T
@BEG_Attrib
3 @RT(0) @RT(0) @RT(0)
@END_Attrib
1 0 @F @F @F @F

@Var @RT(5)sFind @RT(0) @T @F @DT @RT(10)STRING(32) @RT(0) @T @T @STRING 0 @F @RT(2)32 @F
@F @F
@T
@BEG_Attrib
3 @RT(0) @RT(0) @RT(0)
@END_Attrib
1 0 @F @F @F @F

@END_Dcl

@END_Export

@BEG_Export

@BEG_Algo
@POSTUPDATE_ALGORITHM @RT(9)pActivate @STRUCTURED_TEXT
@RT(0) @RT(23)sv_bRemoteMaintActivate @RT(7)TaskVis @F @F
@END_Algo

@BEG_Dcl
@RT(16)DclTreeContainer
3
@Var @RT(18)bRemoteMaintActive @RT(0) @T @T @RENAMED 0 @T @T @DT @RT(4)BOOL @RT(0) @T @T @BASIC 0 @F
@F @F
@T
@BEG_Attrib
3 @RT(0) @RT(0) @RT(0)
@END_Attrib
1 0 @F @F @F @F

@Var @RT(8)SysState @RT(0) @T @T @DERIVED 0 @T @T @DT @RT(15)KSYS_BPApiState @RT(0) @T @T @UNKNOWN 0 @F
@F @F
@T
@BEG_Attrib
3 @RT(0) @RT(0) @RT(0)
@END_Attrib
1 0 @F @F @F @F

@Var @RT(5)dummy @RT(0) @T @F @DT @RT(4)DINT @RT(0) @T @T @BASIC 0 @F
@F @F
@T
@BEG_Attrib
3 @RT(0) @RT(0) @RT(0)
@END_Attrib
1 0 @F @F @F @F

@END_Dcl

@END_Export

@BEG_Body
@TL(38)
(**************************************** WARNING ********************************************
 *** The KEBA Kemro K2 System including software is not intended for safety control tasks! ***
 ***                       For further information see Comment tab!                        ***
 *********************************************************************************************)

SysState := KSYS_BPAPI_VAR_READ('SYS.SERVICES.RemoteMaintenance.Secomea.Sitemanager.status', sTmp);
IF(SysState = cKSYS_BPApiStateOk) THEN
   sv_SiteManager.sState := sTmp;
ELSIF(sv_TraceLevel.bApplication) THEN
   dummy := Print("Remote maintenance: Site manager status cant be read");
END_IF;

SysState := KSYS_BPAPI_VAR_TXTREAD('SYS.SERVICES.RemoteMaintenance.Secomea.Sitemanager.color', sTmp);
IF(SysState = cKSYS_BPApiStateOk) THEN
   sTmp := TOLOWER(sTmp);
   sv_SiteManager.sColor := sTmp;

   // currently the modem status can only be determined with the status string returned
   IF(sTmp = 'red') THEN
      sv_SiteManager.iState := 1;
   ELSIF(sTmp = 'yellow') THEN
      sv_SiteManager.iState := 2;
   ELSIF(sTmp = 'green') THEN
      sv_SiteManager.iState := 3;
   ELSIF(sTmp = 'blue') THEN
      sv_SiteManager.iState := 4;
   ELSE
      sv_SiteManager.iState := 0;
   END_IF;

   sv_SiteManager.bConnected := (sv_SiteManager.iState = 4);

ELSIF(sv_TraceLevel.bApplication) THEN
   dummy := Print("Remote maintenance: Site manager color cant be read");
   sv_SiteManager.bConnected := FALSE;
END_IF;

@END_Body

@@@BEG_Comment@@@
@TL(0)

@@@END_Comment@@@

@BEG_Body
@TL(29)
(**************************************** WARNING ********************************************
 *** The KEBA Kemro K2 System including software is not intended for safety control tasks! ***
 ***                       For further information see Comment tab!                        ***
 *********************************************************************************************)

SysState := KSYS_BPAPI_VAR_TXTREAD('SYS.CFG.Secomea.Sitemanager.Server', sTmp);
IF(SysState = cKSYS_BPApiStateOk) THEN
   sv_SiteManager.sServer := sTmp;
ELSIF(sv_TraceLevel.bApplication) THEN
   dummy := Print("Remote maintenance: Site manager server cant be read");
END_IF;

SysState := KSYS_BPAPI_VAR_TXTREAD('SYS.CFG.Secomea.Sitemanager.Name', sTmp);
IF(SysState = cKSYS_BPApiStateOk) THEN
   sv_SiteManager.sName := sTmp;
ELSIF(sv_TraceLevel.bApplication) THEN
   dummy := Print("Remote maintenance: Site manager name cant be read");
END_IF;

SysState := KSYS_BPAPI_VAR_TXTREAD('SYS.CFG.Secomea.Sitemanager.Domain', sTmp);
IF(SysState = cKSYS_BPApiStateOk) THEN
   sv_SiteManager.sDomain := sTmp;
ELSIF(sv_TraceLevel.bApplication) THEN
   dummy := Print("Remote maintenance: Site manager domain cant be read");
END_IF;

@END_Body

@@@BEG_Comment@@@
@TL(0)

@@@END_Comment@@@

@BEG_Body
@TL(60)
(**************************************** WARNING ********************************************
 *** The KEBA Kemro K2 System including software is not intended for safety control tasks! ***
 ***                       For further information see Comment tab!                        ***
 *********************************************************************************************)

t := GET_RUNTIME();

IF iStep = 0 THEN
   fbTimer(IN := FALSE, PT := t#500ms);
   iStep := 1;
END_IF;

IF iStep = 1 THEN
   fbTimer(IN := TRUE);
   IF(fbTimer.Q) THEN
      iStep := 5;
   END_IF;
END_IF;

IF iStep = 5 THEN
   SysState := KSYS_BPAPI_VAR_READ('SYS.SERVICES.RemoteMaintenance.Secomea.state', iRemoteMaintState);
   IF(SysState <> cKSYS_BPApiStateOk) THEN
      IF(sv_TraceLevel.bApplication) THEN
         dummy := Print("Remote maintenance service not found, KSYS_BPApiState %x", SysState);
      END_IF;
      sv_bRemoteMaintAvailable := FALSE;
      STOP_PROCESS_ALGORITHM(paRun);
      RETURN;
   END_IF;

   IF iRemoteMaintState <> 0 THEN
      // continuously poll for the connection status if the state is active
      // IEC does not have a method for post-updating a BPAPI variable
      aReadSiteManagerStatus();
   ELSIF sv_iRemoteMaintState <> 0 THEN
      // reset the connection status
      IF(sv_SiteManager.sState <> 'disabled') THEN
         sv_SiteManager.sState := 'disabled';
      END_IF;
      IF(sv_SiteManager.sColor <> '') THEN
         sv_SiteManager.sColor := '';
         sv_SiteManager.iState := 0;
      END_IF;
      sv_SiteManager.bConnected := FALSE;
   END_IF;

   sv_iRemoteMaintState := iRemoteMaintState;

   fbTimer(IN := FALSE);
   iStep := 0;
END_IF;

t := GET_RUNTIME() - t;
iTime := LINT_TO_DINT(TIME_TO_LINT(t) / 1000);
IF(iTime >= 10 AND sv_TraceLevel.bApplication) THEN
   dummy := Print("Remote maintenance: Runtime of ABRemoteMaintenance.paRun %d ms", iTime);
END_IF;

@END_Body

@@@BEG_Comment@@@
@TL(0)

@@@END_Comment@@@

@BEG_Body
@TL(24)
(**************************************** WARNING ********************************************
 *** The KEBA Kemro K2 System including software is not intended for safety control tasks! ***
 ***                       For further information see Comment tab!                        ***
 *********************************************************************************************)

IF (NOT mbInit) THEN
   RETURN;
END_IF;

IF(sv_bRemoteMaintAvailable) THEN
   SysState := KSYS_BPAPI_VAR_WRITE('SYS.CFG.Secomea.Sitemanager.Server', sv_sSiteManagerSetServer);
   IF(SysState <> cKSYS_BPApiStateOk) THEN
      dummy := Print("Remote maintenance: Could not set site manager server, KSYS_BPApiState %x", SysState);
      sv_bRemoteMaintActivate := FALSE;
   END_IF;

   aReadSiteManagerServer();

END_IF;

@END_Body

@@@BEG_Comment@@@
@TL(0)

@@@END_Comment@@@

@BEG_Body
@TL(26)
(**************************************** WARNING ********************************************
 *** The KEBA Kemro K2 System including software is not intended for safety control tasks! ***
 ***                       For further information see Comment tab!                        ***
 *********************************************************************************************)

IF (NOT mbInit) THEN
   RETURN;
END_IF;

IF(sv_bRemoteMaintAvailable) THEN

   sTmp := CONCAT(LINT_TO_STRING(sv_iCpuId), '_', sv_sSiteManagerSetName);
   SysState := KSYS_BPAPI_VAR_WRITE('SYS.CFG.Secomea.Sitemanager.Name', sTmp);
   IF(SysState <> cKSYS_BPApiStateOk) THEN
      dummy := Print("Remote maintenance: Could not set site manager name, KSYS_BPApiState %x", SysState);
      sv_bRemoteMaintActivate := FALSE;
   END_IF;

   aReadSiteManagerServer();

END_IF;

@END_Body

@@@BEG_Comment@@@
@TL(0)

@@@END_Comment@@@

@BEG_Body
@TL(83)
(**************************************** WARNING ********************************************
 *** The KEBA Kemro K2 System including software is not intended for safety control tasks! ***
 ***                       For further information see Comment tab!                        ***
 *********************************************************************************************)

HandleData := KCAT_GetHandle('UOS.System');
IF HandleData.Status = KCAT_Status_OK THEN
   Status := KCAT_GetValue(Handle := HandleData.Handle, Buffer := sTemp);
   IF (sTemp = 'Linux') THEN
      bLinux := TRUE;
   END_IF;
END_IF;

IF(NOT bLinux) THEN
   // do not create the nodes on VxWorks - this info does not exist
   // stop and return
   sv_bRemoteMaintAvailable := FALSE;
   STOP_PROCESS_ALGORITHM(paRun);
   RETURN;
END_IF;

// check if RemoteMaintenance software unit is present
SysState := KSYS_BPAPI_VAR_READ('SYS.SERVICES.RemoteMaintenance.Secomea.state', iRemoteMaintState);
IF(SysState <> cKSYS_BPApiStateOk) THEN
   IF(sv_TraceLevel.bApplication) THEN
      dummy := Print("Remote maintenance: service/state not found - stopping, KSYS_BPApiState %x", SysState);
   END_IF;
   // stop and return
   sv_bRemoteMaintAvailable := FALSE;
   STOP_PROCESS_ALGORITHM(paRun);
   RETURN;
END_IF;

// Domain must also be configured
SysState := KSYS_BPAPI_VAR_READ('SYS.CFG.Secomea.Sitemanager.Domain', sSecomeaDomain);
IF(SysState <> cKSYS_BPApiStateOk) THEN
   IF(sv_TraceLevel.bApplication) THEN
      dummy := Print("Remote maintenance: service/domain not found - stopping, KSYS_BPApiState %x", SysState);
   END_IF;
   // stop and return
   sv_bRemoteMaintAvailable := FALSE;
   STOP_PROCESS_ALGORITHM(paRun);
   RETURN;
END_IF;

SysState := KSYS_BPAPI_VAR_READ('SYS.SERVICES.RemoteMaintenance.Secomea.activated', bRemoteMaintActive);
IF(SysState <> cKSYS_BPApiStateOk) THEN
   dummy := Print("Remote maintenance: activated flag not found - setting ignored, KSYS_BPApiState %x", SysState);
   RETURN;
END_IF;
sv_bRemoteMaintActivated := bRemoteMaintActive;
b := WRITE_SV_DIRECT(sv_bRemoteMaintActivate, bRemoteMaintActive);

aReadSiteManagerStatus();
aReadSiteManagerServer();

// initialize the setter variables
sv_sSiteManagerSetServer := sv_SiteManager.sServer;

// prepend <CPUID>_ to the display string
sFind := CONCAT(LINT_TO_STRING(sv_iCpuId), '_');
iTemp := FIND(sv_SiteManager.sName, sFind);

IF (iTemp = 1) THEN
   sv_sSiteManagerSetName := RIGHT(sv_SiteManager.sName, LEN(sv_SiteManager.sName)- LEN(sFind));
ELSE
   sv_sSiteManagerSetName := sv_SiteManager.sName;
END_IF;

sv_iRemoteMaintState := iRemoteMaintState;

// disable ServiceNet IP-switching per default
sv_SNNetworkConfig.sIP := '';

// RemoteMaintenance is available start polling for status changes
sv_bRemoteMaintAvailable := TRUE;
START_PROCESS_ALGORITHM(paRun);

mbInit := TRUE;

@END_Body

@@@BEG_Comment@@@
@TL(0)

@@@END_Comment@@@

@BEG_Body
@TL(27)
(**************************************** WARNING ********************************************
 *** The KEBA Kemro K2 System including software is not intended for safety control tasks! ***
 ***                       For further information see Comment tab!                        ***
 *********************************************************************************************)

// read the current activation status
SysState := KSYS_BPAPI_VAR_READ('SYS.SERVICES.RemoteMaintenance.Secomea.activated', bRemoteMaintActive);
IF(SysState <> cKSYS_BPApiStateOk) THEN
   dummy := Print("Remote maintenance: activated flag not found - setting ignored, KSYS_BPApiState %x", SysState);
   RETURN;
END_IF;

IF(sv_bRemoteMaintActivate = bRemoteMaintActive) THEN
   sv_bRemoteMaintActivated := bRemoteMaintActive;
   RETURN;
END_IF;

// activate service
SysState := KSYS_BPAPI_VAR_WRITE('SYS.SERVICES.RemoteMaintenance.Secomea.activated', sv_bRemoteMaintActivate);
IF(SysState <> cKSYS_BPApiStateOk) THEN
   dummy := Print("Remote maintenance: activated flag not found - could not set, KSYS_BPApiState %x", SysState);
   sv_bRemoteMaintActivate := FALSE;
   RETURN;
END_IF;

sv_bRemoteMaintActivated := sv_bRemoteMaintActivate;

@END_Body

@@@BEG_Comment@@@
@TL(0)

@@@END_Comment@@@
@END_Body

@END_Contents

(* ---- ABServiceNetCtrl.pu ---- *)
(*
@h    ! WARNING !
@h    The Kemro K2 system (including software) only meets category B according to EN 954-1,
@h    thus it is not intended for usage in safety-relevant control applications in the field
@h    of personal safety (e.g. emergency stop).
@h    To implement potentially necessary safety-relevant control tasks, always use additional
@h    external safety devices that are intended for the particular purpose, and meet the necessary
@h    functional safety.
@h    For further information see EN 954-1 (EN ISO 13849-1) and/or the K2-x00 user manual, chapter
@h    "CE conformity, directives and standards".

This AB controls the service net connection state machine
*)

IMPORT_OVER_LISTFILE
 ASSERT
, KPROT_UserInfoLog
, START_PROCESS_ALGORITHM
, tyContactTo
, tsMachineInfo
, tnConnectionStatus
, tnDialogOption
, ABParser
, ABVersionManager
, FBSendData
, KNETWORK_TcpInit
, KSYS_Status
, KPROT_Status
, FBSNNetworkConfig

END_IMPORT

ALGORITHM_BLOCK ABServiceNetCtrl #DUMMY_EDIT_BLOCK

SYSTEM_VAR
 sv_ContactTo : tyContactTo;
 sv_MachineInformation : tsMachineInfo;
 sv_bInitDone : BOOL (* IEC initialisation is finished (after movement registration) *);
 sv_iContactToIdx : DINT;
 sv_bConnect : BOOL;
 sv_ConnectionStatus : tnConnectionStatus;
 sv_HMIResponse : tnDialogOption;
 sv_bDownloadSIMInfo : BOOL;
END_VAR

SYSTEM_OBJECT
 TaskVis : TASK;
 erNoConnection : ALARM;
 erConnectionReset : ALARM;
 erWrongVersion : ALARM;
 erConnectionClosed : ALARM;
END_OBJECT

VAR
 abParser : ABParser;
 abVersionInfo : ABVersionManager;
 fbSend : FBSendData;
END_VAR

VAR CONSTANT
 cConnectionTimeout : TIME := T#30s;
 cVersionServicenetRequired : DINT := 16#100;
 cVersionServicenetClient : DINT := 16#100;
END_VAR

(*
@h    ! WARNING !
@h    The Kemro K2 system (including software) only meets category B according to EN 954-1,
@h    thus it is not intended for usage in safety-relevant control applications in the field
@h    of personal safety (e.g. emergency stop).
@h    To implement potentially necessary safety-relevant control tasks, always use additional
@h    external safety devices that are intended for the particular purpose, and meet the necessary
@h    functional safety.
@h    For further information see EN 954-1 (EN ISO 13849-1) and/or the K2-x00 user manual, chapter
@h    "CE conformity, directives and standards".

Starts state machine algorithm on connect request
*)

POSTUPDATE_ALGORITHM pConnectChanged ON TaskVis(1) WITH sv_bConnect

#BEGIN_EDIT_BLOCK
(**************************************** WARNING ********************************************
 *** The KEBA Kemro K2 System including software is not intended for safety control tasks! ***
 ***                       For further information see Comment tab!                        ***
 *********************************************************************************************)

IF (sv_bConnect) THEN
    IF (NOT sv_bDownloadSIMInfo) THEN
       START_PROCESS_ALGORITHM(paRun);
    ELSE
      // not allowed, download sim info in progress
       sv_bConnect := FALSE;
    END_IF;
END_IF;

;#END_EDIT_BLOCK END_ALGORITHM

(*
@h    ! WARNING !
@h    The Kemro K2 system (including software) only meets category B according to EN 954-1,
@h    thus it is not intended for usage in safety-relevant control applications in the field
@h    of personal safety (e.g. emergency stop).
@h    To implement potentially necessary safety-relevant control tasks, always use additional
@h    external safety devices that are intended for the particular purpose, and meet the necessary
@h    functional safety.
@h    For further information see EN 954-1 (EN ISO 13849-1) and/or the K2-x00 user manual, chapter
@h    "CE conformity, directives and standards".

state machine algorithm
when user requests a connection to ServiceNet this algorithm establishes a TCP connection
and sends a client connection message to ServiceNet.
ServiceNet responds by sending a message containing a protocol version information and a "
request state" number which is used to activate this state.
ABParser is used to parse the recieved messages, it provides access to the recieved data via
function aGetXXXValue().
ServiceNet is expected to send a message at least all 30s, otherwise the connection will be closed.
In case of any error (parsing error, timeout, tcp error, ...) the state changes to "Disconnected"
and the algorithm is stopped.

*)

PROCESS_ALGORITHM paRun ON TaskVis AUTOSTART

VAR
 fbTCPInit : KNETWORK_TcpInit;
 iTmpVal : DINT;
 iRequestState : DINT;
 piTmp : REFTO DINT;
 s : KSYS_Status;
 ILogState : KPROT_Status;
 fbSNNetConfig : FBSNNetworkConfig;
END_VAR

(* IecGraph-Code *)

(* init step *)
INITIAL_STEP S_Init:
AInit (P);
END_STEP

ACTION AInit: #BEGIN_EDIT_BLOCK
// if it is a kvb system wait until initialisation is
// finished in order to get kvb version info which will be
// init is finished if sv_MaskID > cMaskNone (0x10000)
// other version infos are available after sv_bInitDone

piTmp := GET_SYNC_REFTO('KVB.sv_MaskID', T#0s, s);

;#END_EDIT_BLOCK END_ACTION (*AInit*)

(* steps *)
STEP S_ReadVersionInfo:
AReadVersionInfo (P);
END_STEP

ACTION AReadVersionInfo: #BEGIN_EDIT_BLOCK
abVersionInfo.aReadAllVersionInfos();
STOP_PROCESS_ALGORITHM();

;#END_EDIT_BLOCK END_ACTION (*AReadVersionInfo*)
STEP S_NetworkConfigSN:
AInitVars (P);
ANetworkConfigSN (P);
END_STEP

ACTION AInitVars: #BEGIN_EDIT_BLOCK
// initialize variables
sv_HMIResponse := nWaiting;
sv_ConnectionStatus := nConnecting;

;#END_EDIT_BLOCK END_ACTION (*AInitVars*)
ACTION ANetworkConfigSN: #BEGIN_EDIT_BLOCK
fbSNNetConfig(UseServiceNetConfig := TRUE);

;#END_EDIT_BLOCK END_ACTION (*ANetworkConfigSN*)
STEP S_TCPInit:
ATCPInit (N);
ATCPReset (P);
END_STEP

ACTION ATCPInit: #BEGIN_EDIT_BLOCK
// connect TCP socket
fbTCPInit( Execute := TRUE,
          RemoteIP := sv_ContactTo[sv_iContactToIdx].sAddress,
          RemotePort := cServiceNet_PortNumber);

;#END_EDIT_BLOCK END_ACTION (*ATCPInit*)
ACTION ATCPReset: #BEGIN_EDIT_BLOCK
ILogState := KPROT_UserInfoLog('ServiceNet state: %5s', 0, 0, 0, 0, 'connecting');

;#END_EDIT_BLOCK END_ACTION (*ATCPReset*)
STEP S_TCPInitError:
ATCPInitError (N);
END_STEP

ACTION ATCPInitError: #BEGIN_EDIT_BLOCK
SET_ALARM(Name := erNoConnection,
              Param1 := sv_ContactTo[sv_iContactToIdx].sAddress);

;#END_EDIT_BLOCK END_ACTION (*ATCPInitError*)
STEP S_Connecting:
AReset (P);
AConnecting (N);
ACommunication (S);
END_STEP

ACTION AReset: #BEGIN_EDIT_BLOCK
RESET_ALARM(erNoConnection);
RESET_ALARM(erConnectionReset);
RESET_ALARM(erWrongVersion);
RESET_ALARM(erConnectionClosed);

abParser.aGetDINTValue(Execute := FALSE);
fbSend(FALSE, fbTCPInit.TcpHdl, cVersionServicenetClient, abVersionInfo);

;#END_EDIT_BLOCK END_ACTION (*AReset*)
ACTION AConnecting: #BEGIN_EDIT_BLOCK
// check ServiceNet version
abParser.aGetDINTValue(TRUE, "VersionServiceNet", iTmpVal);

// ServiceNet version to old, newer version required -> alarm and disconnect
IF (abParser.aGetDINTValue.bFound AND (iTmpVal < cVersionServicenetRequired)) THEN
    SET_ALARM(Name := erWrongVersion,
            Param1 := REAL_TO_FORMATTED_STRING(INT_TO_REAL(BCD_TO_INT(DINT_TO_WORD(cVersionServicenetRequired))) / 100.0, 2, 2),
            Param2 := REAL_TO_FORMATTED_STRING(INT_TO_REAL(BCD_TO_INT(DINT_TO_WORD(iTmpVal))) / 100.0, 2, 2)
             );
    sv_bConnect := FALSE; // exit transition
END_IF;

;#END_EDIT_BLOCK END_ACTION (*AConnecting*)
ACTION ACommunication: #BEGIN_EDIT_BLOCK
// parse received messages, reset SFC in case of an Error
abParser.aParse(Execute := TRUE,
                TcpHdl := fbTCPInit.TcpHdl);

// check connection timeout
IF (abParser.aParse.ElapsedTimeSinceLastObj > cConnectionTimeout) THEN
    SET_ALARM(Name := erConnectionReset, Param1 := 1);
    sv_bConnect := FALSE;  // exit transition
ELSIF (abParser.aParse.Error) THEN
    SET_ALARM(Name := erConnectionReset, Param1 := 2);
    sv_bConnect := FALSE;  // exit transition
END_IF;

// send message, reset SFC in case of an error
fbSend(Execute := TRUE);
IF (fbSend.Error) THEN
    SET_ALARM(Name := erConnectionReset, Param1 := 3);
    sv_bConnect := FALSE; // exit transition
END_IF;

;#END_EDIT_BLOCK END_ACTION (*ACommunication*)
STEP S_GetReqState:
AReset2 (P);
AGetRequestState (S);
END_STEP

ACTION AReset2: #BEGIN_EDIT_BLOCK
abParser.aGetDINTValue(Execute := FALSE);

;#END_EDIT_BLOCK END_ACTION (*AReset2*)
ACTION AGetRequestState: #BEGIN_EDIT_BLOCK
// cyclic update of local variable iRequestState
abParser.aGetDINTValue(TRUE, "RequestState", iRequestState);

;#END_EDIT_BLOCK END_ACTION (*AGetRequestState*)
STEP S_RequestPending:
ARequestPending (P);
END_STEP

ACTION ARequestPending: #BEGIN_EDIT_BLOCK
sv_ConnectionStatus := nRequestPending;
ILogState := KPROT_UserInfoLog('ServiceNet state: %5s', 0, 0, 0, 0, 'request pending');

;#END_EDIT_BLOCK END_ACTION (*ARequestPending*)
STEP S_ServiceAccepted:
AServiceAccepted (P);
END_STEP

ACTION AServiceAccepted: #BEGIN_EDIT_BLOCK
sv_ConnectionStatus := nServiceAccepted;
ILogState := KPROT_UserInfoLog('ServiceNet state: %5s', 0, 0, 0, 0, 'service accepted');

;#END_EDIT_BLOCK END_ACTION (*AServiceAccepted*)
STEP S_ServiceAccessRequest:
AServiceAccessRequest (P);
END_STEP

ACTION AServiceAccessRequest: #BEGIN_EDIT_BLOCK
sv_HMIResponse := nWaiting;
sv_ConnectionStatus := nServiceAccessRequest;
ILogState := KPROT_UserInfoLog('ServiceNet state: %5s', 0, 0, 0, 0, 'service access request');

;#END_EDIT_BLOCK END_ACTION (*AServiceAccessRequest*)
STEP S_ServiceActive:
AServiceActive (P);
END_STEP

ACTION AServiceActive: #BEGIN_EDIT_BLOCK
sv_ConnectionStatus := nServiceActive;
ILogState := KPROT_UserInfoLog('ServiceNet state: %5s', 0, 0, 0, 0, 'service active');

;#END_EDIT_BLOCK END_ACTION (*AServiceActive*)
STEP S_Disconnecting:
ACommunication (R);
AGetRequestState (R);
AResetParser (P);
ADisconnect (N);
END_STEP

ACTION AResetParser: #BEGIN_EDIT_BLOCK
abParser.aParse(Execute := FALSE);
ILogState := KPROT_UserInfoLog('ServiceNet state: %5s', 0, 0, 0, 0, 'disconnected');

;#END_EDIT_BLOCK END_ACTION (*AResetParser*)
ACTION ADisconnect: #BEGIN_EDIT_BLOCK
IF (iRequestState = cREQSTATE_SERVICE_CLOSE) THEN
   // ServiceNet has sent disconnect command
   SET_ALARM(erConnectionClosed);
END_IF;

fbTCPInit(Execute := FALSE);
fbSNNetConfig(UseServiceNetConfig := FALSE);

iRequestState := 0;
sv_ConnectionStatus := nDisconnected;
sv_bConnect := FALSE;
STOP_PROCESS_ALGORITHM();

;#END_EDIT_BLOCK END_ACTION (*ADisconnect*)
STEP S_Disconnected:
END_STEP

(* transitions *)
GO_ON_TRANSITION Trans15 (* Trans15 *) FROM S_Init TO S_ReadVersionInfo :=  #BEGIN_EDIT_BLOCK
((piTmp = EMPTY) OR (piTmp^ > 16#10000)) AND sv_bInitDone
;#END_EDIT_BLOCK
END_TRANSITION

TRANSITION Trans29 (* Trans29 *) FROM S_ReadVersionInfo TO S_NetworkConfigSN :=  #BEGIN_EDIT_BLOCK
TRUE
;#END_EDIT_BLOCK
END_TRANSITION

TRANSITION Trans40 (* Trans40 *) FROM S_NetworkConfigSN TO S_TCPInit :=  #BEGIN_EDIT_BLOCK
NOT fbSNNetConfig.Error
;#END_EDIT_BLOCK
END_TRANSITION

TRANSITION Trans41 (* Trans41 *) FROM S_NetworkConfigSN TO S_TCPInitError :=  #BEGIN_EDIT_BLOCK
fbSNNetConfig.Error
;#END_EDIT_BLOCK
END_TRANSITION

GO_ON_TRANSITION Trans2 (* Trans2 *) FROM S_TCPInit TO S_Connecting :=  #BEGIN_EDIT_BLOCK
fbTCPInit.Done
;#END_EDIT_BLOCK
END_TRANSITION

GO_ON_TRANSITION Trans33 (* Trans33 *) FROM S_TCPInit TO S_TCPInitError :=  #BEGIN_EDIT_BLOCK
fbTCPInit.Error
;#END_EDIT_BLOCK
END_TRANSITION

GO_ON_TRANSITION Trans34 (* Trans34 *) FROM S_TCPInitError TO S_Disconnecting :=  #BEGIN_EDIT_BLOCK
TRUE
;#END_EDIT_BLOCK
END_TRANSITION

GO_ON_TRANSITION Trans39 (* Trans39 *) FROM S_TCPInit TO S_Disconnecting :=  #BEGIN_EDIT_BLOCK
NOT sv_bConnect
;#END_EDIT_BLOCK
END_TRANSITION

GO_ON_TRANSITION Trans13 (* Trans13 *) FROM S_Connecting TO S_GetReqState :=  #BEGIN_EDIT_BLOCK
abParser.aGetDINTValue.bFound AND (NOT (iTmpVal < cVersionServicenetRequired))
;#END_EDIT_BLOCK
END_TRANSITION

GO_ON_TRANSITION Trans22 (* Trans22 *) FROM S_GetReqState TO S_RequestPending :=  #BEGIN_EDIT_BLOCK
abParser.aGetDINTValue.bFound AND (iRequestState >= cREQSTATE_SERVICE_REQPENDING)
;#END_EDIT_BLOCK
END_TRANSITION

GO_ON_TRANSITION Trans14 (* Trans14 *) FROM S_RequestPending TO S_ServiceAccepted :=  #BEGIN_EDIT_BLOCK
iRequestState >= cREQSTATE_SERVICE_ACCEPTED
;#END_EDIT_BLOCK
END_TRANSITION

GO_ON_TRANSITION Trans16 (* Trans16 *) FROM S_ServiceAccepted TO S_ServiceAccessRequest :=  #BEGIN_EDIT_BLOCK
iRequestState >= cREQSTATE_SERVICE_ACCESSREQ
;#END_EDIT_BLOCK
END_TRANSITION

GO_ON_TRANSITION Trans17 (* Trans17 *) FROM S_ServiceAccessRequest TO S_Disconnecting :=  #BEGIN_EDIT_BLOCK
sv_HMIResponse = nNo
;#END_EDIT_BLOCK
END_TRANSITION

GO_ON_TRANSITION Trans26 (* Trans26 *) FROM S_ServiceAccessRequest TO S_ServiceActive :=  #BEGIN_EDIT_BLOCK
sv_HMIResponse = nYes
;#END_EDIT_BLOCK
END_TRANSITION

GO_ON_TRANSITION Trans23 (* Trans23 *) FROM S_ServiceActive TO S_Disconnecting :=  #BEGIN_EDIT_BLOCK
iRequestState = cREQSTATE_SERVICE_CLOSE  // ServiceNet wants to disconnect
;#END_EDIT_BLOCK
END_TRANSITION

GO_ON_TRANSITION Trans38 (* Trans38 *) FROM S_Disconnecting TO S_Disconnected :=  #BEGIN_EDIT_BLOCK
TRUE
;#END_EDIT_BLOCK
END_TRANSITION

TRANSITION Trans25 (* Trans25 *) FROM S_Disconnected TO S_NetworkConfigSN :=  #BEGIN_EDIT_BLOCK
sv_bConnect
;#END_EDIT_BLOCK
END_TRANSITION

(* end IecGraph-Code *)
(* sfc-code *)

(* exits *)

EXIT_TRANSITION TDisconnectClient := #BEGIN_EDIT_BLOCK
(S_Init.X = FALSE)
AND (S_ReadVersionInfo.X = FALSE)
AND (S_TCPInit.X = FALSE)
AND (S_Disconnecting.X = FALSE)
AND (S_Disconnected.X = FALSE)
AND (sv_bConnect = FALSE)
;#END_EDIT_BLOCK
PRIORITY 1 WITH  INITIAL_STEP S_Disconnecting: END_STEP
END_TRANSITION

EXIT_TRANSITION TDisconnectServer := #BEGIN_EDIT_BLOCK
iRequestState = cREQSTATE_SERVICE_CLOSE
;#END_EDIT_BLOCK
PRIORITY 1 WITH  INITIAL_STEP S_Disconnecting: END_STEP
END_TRANSITION
(* end sfc-code *)

END_ALGORITHM

END_ALGORITHM_BLOCK

#END_OF_IEC_PART

@Puma @IecEditor 6 121 @Pou 25
@@@BEG_Comment@@@
@h    ! WARNING !
@h    The Kemro K2 system (including software) only meets category B according to EN 954-1,
@h    thus it is not intended for usage in safety-relevant control applications in the field
@h    of personal safety (e.g. emergency stop).
@h    To implement potentially necessary safety-relevant control tasks, always use additional
@h    external safety devices that are intended for the particular purpose, and meet the necessary
@h    functional safety.
@h    For further information see EN 954-1 (EN ISO 13849-1) and/or the K2-x00 user manual, chapter
@h    "CE conformity, directives and standards".

This AB controls the service net connection state machine
@@@END_Comment@@@

@BEG_Contents

@BEG_Func
@RT(17)FuncTreeContainer
3
@Var @RT(6)ASSERT @RT(0) @T @T @DERIVED 0 @F @RT(8)FUNCTION @F
@T
@BEG_Attrib
0 @RT(0) @RT(0)
@END_Attrib
1 1 @F @F @F @F

@Var @RT(17)KPROT_UserInfoLog @RT(0) @T @T @DERIVED 0 @F @RT(22)KEBA_STANDARD_FUNCTION @F
@T
@BEG_Attrib
0 @RT(0) @RT(0)
@END_Attrib
1 1 @F @F @F @F

@Var @RT(23)START_PROCESS_ALGORITHM @RT(0) @T @T @DERIVED 0 @F @RT(23)KEBA_STANDARD_PROCEDURE @F
@T
@BEG_Attrib
0 @RT(0) @RT(0)
@END_Attrib
1 1 @F @F @F @F

@END_Func

@BEG_Const
@RT(18)ConstTreeContainer
0
@END_Const

@BEG_Export

@BEG_Kind
@ALGORITHM_BLOCK @RT(16)ABServiceNetCtrl @STRUCTURED_TEXT
@RT(0) @RT(0) @RT(0)
@END_Kind

@BEG_Dcl
@RT(16)DclTreeContainer
19
@Var @RT(12)sv_ContactTo @RT(0) @T @T @DERIVED 0 @T @T @DT @RT(11)tyContactTo @RT(0) @T @T @UNKNOWN 0 @F
@F @F
@T
@BEG_Attrib
3 @RT(0) @RT(0) @RT(0)
@END_Attrib
1 8 @F @F @F @F

@Var @RT(21)sv_MachineInformation @RT(0) @T @T @DERIVED 0 @T @T @DT @RT(13)tsMachineInfo @RT(0) @T @T @UNKNOWN 0 @F
@F @F
@T
@BEG_Attrib
3 @RT(0) @RT(0) @RT(0)
@END_Attrib
1 8 @F @F @F @F

@Var @RT(12)sv_bInitDone @RT(0) @T @F @DT @RT(4)BOOL @RT(0) @T @T @BASIC 0 @F
@F @F
@T
@BEG_Attrib
3 @RT(0) @RT(60)IEC initialisation is finished (after movement registration) @RT(0)
@END_Attrib
1 8 @F @F @F @F

@Var @RT(16)sv_iContactToIdx @RT(0) @T @F @DT @RT(4)DINT @RT(0) @T @T @BASIC 0 @F
@F @F
@T
@BEG_Attrib
3 @RT(0) @RT(0) @RT(0)
@END_Attrib
1 8 @F @F @F @F

@Var @RT(11)sv_bConnect @RT(0) @T @F @DT @RT(4)BOOL @RT(0) @T @T @BASIC 0 @F
@F @F
@T
@BEG_Attrib
3 @RT(0) @RT(0) @RT(0)
@END_Attrib
1 8 @F @F @F @F

@Var @RT(19)sv_ConnectionStatus @RT(0) @T @T @DERIVED 0 @T @T @DT @RT(18)tnConnectionStatus @RT(0) @T @T @UNKNOWN 0 @F
@F @F
@T
@BEG_Attrib
3 @RT(0) @RT(0) @RT(0)
@END_Attrib
1 8 @F @F @F @F

@Var @RT(7)TaskVis @RT(0) @T @T @RENAMED 0 @T @T @DT @RT(4)TASK @RT(0) @T @T @BASIC 0 @F
@F @F
@T
@BEG_Attrib
3 @RT(0) @RT(0) @RT(0)
@END_Attrib
1 7 @F @F @F @F

@Var @RT(14)sv_HMIResponse @RT(0) @T @T @DERIVED 0 @T @T @DT @RT(14)tnDialogOption @RT(0) @T @T @UNKNOWN 0 @F
@F @F
@T
@BEG_Attrib
3 @RT(0) @RT(0) @RT(0)
@END_Attrib
1 8 @F @F @F @F

@Var @RT(18)cConnectionTimeout @RT(0) @T @F @DT @RT(4)TIME @RT(0) @T @T @BASIC 0 @F
@F @F
@T
@BEG_Attrib
3 @RT(5)T#30s @RT(0) @RT(0)
@END_Attrib
1 15 @F @F @F @F

@Var @RT(26)cVersionServicenetRequired @RT(0) @T @F @DT @RT(4)DINT @RT(0) @T @T @BASIC 0 @F
@F @F
@T
@BEG_Attrib
3 @RT(6)16#100 @RT(0) @RT(0)
@END_Attrib
1 15 @F @F @F @F

@Var @RT(24)cVersionServicenetClient @RT(0) @T @F @DT @RT(4)DINT @RT(0) @T @T @BASIC 0 @F
@F @F
@T
@BEG_Attrib
3 @RT(6)16#100 @RT(0) @RT(0)
@END_Attrib
1 15 @F @F @F @F

@Var @RT(8)abParser @RT(0) @T @T @DERIVED 0 @T @T @DT @RT(8)ABParser @RT(0) @T @T @UNKNOWN 0 @F
@F @F
@T
@BEG_Attrib
3 @RT(0) @RT(0) @RT(0)
@END_Attrib
1 0 @F @F @F @F

@Var @RT(14)erNoConnection @RT(0) @T @F @DT @RT(5)ALARM @RT(0) @T @T @BASIC 0 @F
@F @F
@T
@BEG_Attrib
3 @RT(0) @RT(0) @RT(0)
@END_Attrib
1 7 @F @F @F @F

@Var @RT(17)erConnectionReset @RT(0) @T @F @DT @RT(5)ALARM @RT(0) @T @T @BASIC 0 @F
@F @F
@T
@BEG_Attrib
3 @RT(0) @RT(0) @RT(0)
@END_Attrib
1 7 @F @F @F @F

@Var @RT(14)erWrongVersion @RT(0) @T @F @DT @RT(5)ALARM @RT(0) @T @T @BASIC 0 @F
@F @F
@T
@BEG_Attrib
3 @RT(0) @RT(0) @RT(0)
@END_Attrib
1 7 @F @F @F @F

@Var @RT(18)erConnectionClosed @RT(0) @T @F @DT @RT(5)ALARM @RT(0) @T @T @BASIC 0 @F
@F @F
@T
@BEG_Attrib
3 @RT(0) @RT(0) @RT(0)
@END_Attrib
1 7 @F @F @F @F

@Var @RT(13)abVersionInfo @RT(0) @T @T @DERIVED 0 @T @T @DT @RT(16)ABVersionManager @RT(0) @T @T @UNKNOWN 0 @F
@F @F
@T
@BEG_Attrib
3 @RT(0) @RT(0) @RT(0)
@END_Attrib
1 0 @F @F @F @F

@Var @RT(19)sv_bDownloadSIMInfo @RT(0) @T @F @DT @RT(4)BOOL @RT(0) @T @T @BASIC 0 @F
@F @F
@T
@BEG_Attrib
3 @RT(0) @RT(0) @RT(0)
@END_Attrib
1 8 @F @F @F @F

@Var @RT(6)fbSend @RT(0) @T @T @DERIVED 0 @T @T @DT @RT(10)FBSendData @RT(0) @T @T @UNKNOWN 0 @F
@F @F
@T
@BEG_Attrib
3 @RT(0) @RT(0) @RT(0)
@END_Attrib
1 0 @F @F @F @F

@END_Dcl

@END_Export

@BEG_Body

2

@BEG_Export

@BEG_Algo
@POSTUPDATE_ALGORITHM @RT(15)pConnectChanged @STRUCTURED_TEXT
@RT(0) @RT(11)sv_bConnect @RT(10)TaskVis(1) @F @F
@END_Algo

@BEG_Dcl
@RT(16)DclTreeContainer
0
@END_Dcl

@END_Export

@BEG_Export

@BEG_Algo
@PROCESS_ALGORITHM @RT(5)paRun @SEQUENTIAL_FLOW_CHART
@RT(0) @RT(0) @RT(7)TaskVis @T @F
@END_Algo

@BEG_Dcl
@RT(16)DclTreeContainer
7
@Var @RT(9)fbTCPInit @RT(0) @T @T @DERIVED 0 @T @T @DT @RT(16)KNETWORK_TcpInit @RT(0) @T @T @UNKNOWN 0 @F
@F @F
@T
@BEG_Attrib
3 @RT(0) @RT(0) @RT(0)
@END_Attrib
1 0 @F @F @F @F

@Var @RT(7)iTmpVal @RT(0) @T @F @DT @RT(4)DINT @RT(0) @T @T @BASIC 0 @F
@F @F
@T
@BEG_Attrib
3 @RT(0) @RT(0) @RT(0)
@END_Attrib
1 0 @F @F @F @F

@Var @RT(13)iRequestState @RT(0) @T @F @DT @RT(4)DINT @RT(0) @T @T @BASIC 0 @F
@F @F
@T
@BEG_Attrib
3 @RT(0) @RT(0) @RT(0)
@END_Attrib
1 0 @F @F @F @F

@Var @RT(5)piTmp @RT(0) @T @T @REFTO 0 @T @DT @RT(4)DINT @RT(0) @T @T @BASIC 0 @F
@F @F
@T
@BEG_Attrib
3 @RT(0) @RT(0) @RT(0)
@END_Attrib
1 0 @F @F @F @F

@Var @RT(1)s @RT(0) @T @T @DERIVED 0 @T @T @DT @RT(11)KSYS_Status @RT(0) @T @T @UNKNOWN 0 @F
@F @F
@T
@BEG_Attrib
3 @RT(0) @RT(0) @RT(0)
@END_Attrib
1 0 @F @F @F @F

@Var @RT(9)ILogState @RT(0) @T @T @RENAMED 0 @T @T @DT @RT(12)KPROT_Status @RT(0) @T @T @UNKNOWN 0 @F
@F @F
@T
@BEG_Attrib
3 @RT(0) @RT(0) @RT(0)
@END_Attrib
1 0 @F @F @F @F

@Var @RT(13)fbSNNetConfig @RT(0) @T @T @DERIVED 0 @T @T @DT @RT(17)FBSNNetworkConfig @RT(0) @T @T @UNKNOWN 0 @F
@F @F
@T
@BEG_Attrib
3 @RT(0) @RT(0) @RT(0)
@END_Attrib
1 0 @F @F @F @F

@END_Dcl

@END_Export

@BEG_Body
@TL(16)
(**************************************** WARNING ********************************************
 *** The KEBA Kemro K2 System including software is not intended for safety control tasks! ***
 ***                       For further information see Comment tab!                        ***
 *********************************************************************************************)

IF (sv_bConnect) THEN
    IF (NOT sv_bDownloadSIMInfo) THEN
       START_PROCESS_ALGORITHM(paRun);
    ELSE
      // not allowed, download sim info in progress
       sv_bConnect := FALSE;
    END_IF;
END_IF;

@END_Body

@@@BEG_Comment@@@
@TL(11)
@h    ! WARNING !
@h    The Kemro K2 system (including software) only meets category B according to EN 954-1,
@h    thus it is not intended for usage in safety-relevant control applications in the field
@h    of personal safety (e.g. emergency stop).
@h    To implement potentially necessary safety-relevant control tasks, always use additional
@h    external safety devices that are intended for the particular purpose, and meet the necessary
@h    functional safety.
@h    For further information see EN 954-1 (EN ISO 13849-1) and/or the K2-x00 user manual, chapter
@h    "CE conformity, directives and standards".

Starts state machine algorithm on connect request
@@@END_Comment@@@

@BEG_SfcBody
54 34 51

@BEG_SfcData 2
@StepSeq @RT(4)sseq @F 5
@Step @RT(6)S_Init @F @T @F @F @RT(0) @F
@AcbCont @RT(7)unnamed @F 1
@Acb @RT(5)AInit @F @T @RT(1)P @RT(0) @F @F @T @TL(7)
// if it is a kvb system wait until initialisation is
// finished in order to get kvb version info which will be
// init is finished if sv_MaskID > cMaskNone (0x10000)
// other version infos are available after sv_bInitDone

piTmp := GET_SYNC_REFTO('KVB.sv_MaskID', T#0s, s);

@F

@Trans @RT(7)Trans15 @F @T @F @F @T @F @TL(2)
((piTmp = EMPTY) OR (piTmp^ > 16#10000)) AND sv_bInitDone

@RT(7)Trans15 @F
@Step @RT(17)S_ReadVersionInfo @F @F @F @F @RT(0) @F
@AcbCont @RT(7)unnamed @F 1
@Acb @RT(16)AReadVersionInfo @F @T @RT(1)P @RT(0) @F @F @T @TL(3)
abVersionInfo.aReadAllVersionInfos();
STOP_PROCESS_ALGORITHM();

@F

@Trans @RT(7)Trans29 @F @T @F @F @T @T @TL(2)
TRUE

@RT(7)Trans29 @F
@Loop @RT(4)loop @F 2
@StepSeq @RT(3)seq @F 17
@Step @RT(17)S_NetworkConfigSN @F @F @F @F @RT(0) @F
@AcbCont @RT(7)unnamed @F 2
@Acb @RT(9)AInitVars @F @T @RT(1)P @RT(0) @F @F @T @TL(4)
// initialize variables
sv_HMIResponse := nWaiting;
sv_ConnectionStatus := nConnecting;

@F
@Acb @RT(16)ANetworkConfigSN @F @T @RT(1)P @RT(0) @F @F @T @TL(2)
fbSNNetConfig(UseServiceNetConfig := TRUE);

@F

@AltBranch @RT(3)alt @F 2
@TransSeq @RT(4)tseq @F 1
@Trans @RT(7)Trans40 @F @T @F @F @T @T @TL(2)
NOT fbSNNetConfig.Error

@RT(7)Trans40 @F

@TransSeq @RT(4)tseq @F 2
@Trans @RT(7)Trans41 @F @T @F @F @T @T @TL(2)
fbSNNetConfig.Error

@RT(7)Trans41 @F
@Goto @RT(14)S_TCPInitError @F @F

@Step @RT(9)S_TCPInit @F @F @F @F @RT(0) @F
@AcbCont @RT(7)unnamed @F 2
@Acb @RT(8)ATCPInit @F @T @RT(1)N @RT(0) @F @F @T @TL(5)
// connect TCP socket
fbTCPInit( Execute := TRUE,
          RemoteIP := sv_ContactTo[sv_iContactToIdx].sAddress,
          RemotePort := cServiceNet_PortNumber);

@F
@Acb @RT(9)ATCPReset @F @T @RT(1)P @RT(0) @F @F @T @TL(2)
ILogState := KPROT_UserInfoLog('ServiceNet state: %5s', 0, 0, 0, 0, 'connecting');

@F

@AltBranch @RT(3)alt @F 3
@TransSeq @RT(4)tseq @F 1
@Trans @RT(6)Trans2 @F @T @F @F @T @F @TL(2)
fbTCPInit.Done

@RT(6)Trans2 @F

@TransSeq @RT(4)tseq @F 4
@Trans @RT(7)Trans33 @F @T @F @F @T @F @TL(2)
fbTCPInit.Error

@RT(7)Trans33 @F
@Step @RT(14)S_TCPInitError @F @F @T @F @RT(0) @F
@AcbCont @RT(7)unnamed @F 1
@Acb @RT(13)ATCPInitError @F @T @RT(1)N @RT(0) @F @F @T @TL(3)
SET_ALARM(Name := erNoConnection,
              Param1 := sv_ContactTo[sv_iContactToIdx].sAddress);

@F

@Trans @RT(7)Trans34 @F @T @F @F @T @F @TL(2)
TRUE

@RT(7)Trans34 @F
@Goto @RT(15)S_Disconnecting @F @F

@TransSeq @RT(4)tseq @F 2
@Trans @RT(7)Trans39 @F @T @F @F @T @F @TL(2)
NOT sv_bConnect

@RT(7)Trans39 @F
@Goto @RT(15)S_Disconnecting @F @F

@Step @RT(12)S_Connecting @F @F @F @F @RT(0) @F
@AcbCont @RT(7)unnamed @F 3
@Acb @RT(6)AReset @F @T @RT(1)P @RT(0) @F @F @T @TL(8)
RESET_ALARM(erNoConnection);
RESET_ALARM(erConnectionReset);
RESET_ALARM(erWrongVersion);
RESET_ALARM(erConnectionClosed);

abParser.aGetDINTValue(Execute := FALSE);
fbSend(FALSE, fbTCPInit.TcpHdl, cVersionServicenetClient, abVersionInfo);

@F
@Acb @RT(11)AConnecting @F @T @RT(1)N @RT(0) @F @F @T @TL(13)
// check ServiceNet version
abParser.aGetDINTValue(TRUE, "VersionServiceNet", iTmpVal);

// ServiceNet version to old, newer version required -> alarm and disconnect
IF (abParser.aGetDINTValue.bFound AND (iTmpVal < cVersionServicenetRequired)) THEN
    SET_ALARM(Name := erWrongVersion,
            Param1 := REAL_TO_FORMATTED_STRING(INT_TO_REAL(BCD_TO_INT(DINT_TO_WORD(cVersionServicenetRequired))) / 100.0, 2, 2),
            Param2 := REAL_TO_FORMATTED_STRING(INT_TO_REAL(BCD_TO_INT(DINT_TO_WORD(iTmpVal))) / 100.0, 2, 2)
             );
    sv_bConnect := FALSE; // exit transition
END_IF;

@F
@Acb @RT(14)ACommunication @F @T @RT(1)S @RT(0) @F @F @T @TL(21)
// parse received messages, reset SFC in case of an Error
abParser.aParse(Execute := TRUE,
                TcpHdl := fbTCPInit.TcpHdl);

// check connection timeout
IF (abParser.aParse.ElapsedTimeSinceLastObj > cConnectionTimeout) THEN
    SET_ALARM(Name := erConnectionReset, Param1 := 1);
    sv_bConnect := FALSE;  // exit transition
ELSIF (abParser.aParse.Error) THEN
    SET_ALARM(Name := erConnectionReset, Param1 := 2);
    sv_bConnect := FALSE;  // exit transition
END_IF;

// send message, reset SFC in case of an error
fbSend(Execute := TRUE);
IF (fbSend.Error) THEN
    SET_ALARM(Name := erConnectionReset, Param1 := 3);
    sv_bConnect := FALSE; // exit transition
END_IF;

@F

@Trans @RT(7)Trans13 @F @T @F @F @T @F @TL(2)
abParser.aGetDINTValue.bFound AND (NOT (iTmpVal < cVersionServicenetRequired))

@RT(7)Trans13 @F
@Step @RT(13)S_GetReqState @F @F @F @F @RT(0) @F
@AcbCont @RT(7)unnamed @F 2
@Acb @RT(7)AReset2 @F @T @RT(1)P @RT(0) @F @F @T @TL(2)
abParser.aGetDINTValue(Execute := FALSE);

@F
@Acb @RT(16)AGetRequestState @F @T @RT(1)S @RT(0) @F @F @T @TL(3)
// cyclic update of local variable iRequestState
abParser.aGetDINTValue(TRUE, "RequestState", iRequestState);

@F

@Trans @RT(7)Trans22 @F @T @F @F @T @F @TL(2)
abParser.aGetDINTValue.bFound AND (iRequestState >= cREQSTATE_SERVICE_REQPENDING)

@RT(7)Trans22 @F
@Step @RT(16)S_RequestPending @F @F @F @F @RT(0) @F
@AcbCont @RT(7)unnamed @F 1
@Acb @RT(15)ARequestPending @F @T @RT(1)P @RT(0) @F @F @T @TL(3)
sv_ConnectionStatus := nRequestPending;
ILogState := KPROT_UserInfoLog('ServiceNet state: %5s', 0, 0, 0, 0, 'request pending');

@F

@Trans @RT(7)Trans14 @F @T @F @F @T @F @TL(2)
iRequestState >= cREQSTATE_SERVICE_ACCEPTED

@RT(7)Trans14 @F
@Step @RT(17)S_ServiceAccepted @F @F @F @F @RT(0) @F
@AcbCont @RT(7)unnamed @F 1
@Acb @RT(16)AServiceAccepted @F @T @RT(1)P @RT(0) @F @F @T @TL(3)
sv_ConnectionStatus := nServiceAccepted;
ILogState := KPROT_UserInfoLog('ServiceNet state: %5s', 0, 0, 0, 0, 'service accepted');

@F

@Trans @RT(7)Trans16 @F @T @F @F @T @F @TL(2)
iRequestState >= cREQSTATE_SERVICE_ACCESSREQ

@RT(7)Trans16 @F
@Step @RT(22)S_ServiceAccessRequest @F @F @F @F @RT(0) @F
@AcbCont @RT(7)unnamed @F 1
@Acb @RT(21)AServiceAccessRequest @F @T @RT(1)P @RT(0) @F @F @T @TL(4)
sv_HMIResponse := nWaiting;
sv_ConnectionStatus := nServiceAccessRequest;
ILogState := KPROT_UserInfoLog('ServiceNet state: %5s', 0, 0, 0, 0, 'service access request');

@F

@AltBranch @RT(3)alt @F 2
@TransSeq @RT(4)tseq @F 1
@Trans @RT(7)Trans17 @F @T @F @F @T @F @TL(2)
sv_HMIResponse = nNo

@RT(7)Trans17 @F

@TransSeq @RT(4)tseq @F 3
@Trans @RT(7)Trans26 @F @T @F @F @T @F @TL(2)
sv_HMIResponse = nYes

@RT(7)Trans26 @F
@Step @RT(15)S_ServiceActive @F @F @F @F @RT(0) @F
@AcbCont @RT(7)unnamed @F 1
@Acb @RT(14)AServiceActive @F @T @RT(1)P @RT(0) @F @F @T @TL(3)
sv_ConnectionStatus := nServiceActive;
ILogState := KPROT_UserInfoLog('ServiceNet state: %5s', 0, 0, 0, 0, 'service active');

@F

@Trans @RT(7)Trans23 @F @T @F @F @T @F @TL(2)
iRequestState = cREQSTATE_SERVICE_CLOSE  // ServiceNet wants to disconnect

@RT(7)Trans23 @F

@Step @RT(15)S_Disconnecting @F @F @T @F @RT(0) @F
@AcbCont @RT(7)unnamed @F 4
@Acb @RT(14)ACommunication @F @F @RT(1)R @RT(0) @F @F @T @F
@Acb @RT(16)AGetRequestState @F @F @RT(1)R @RT(0) @F @F @T @F
@Acb @RT(12)AResetParser @F @T @RT(1)P @RT(0) @F @F @T @TL(3)
abParser.aParse(Execute := FALSE);
ILogState := KPROT_UserInfoLog('ServiceNet state: %5s', 0, 0, 0, 0, 'disconnected');

@F
@Acb @RT(11)ADisconnect @F @T @RT(1)N @RT(0) @F @F @T @TL(13)
IF (iRequestState = cREQSTATE_SERVICE_CLOSE) THEN
   // ServiceNet has sent disconnect command
   SET_ALARM(erConnectionClosed);
END_IF;

fbTCPInit(Execute := FALSE);
fbSNNetConfig(UseServiceNetConfig := FALSE);

iRequestState := 0;
sv_ConnectionStatus := nDisconnected;
sv_bConnect := FALSE;
STOP_PROCESS_ALGORITHM();

@F

@Trans @RT(7)Trans38 @F @T @F @F @T @F @TL(2)
TRUE

@RT(7)Trans38 @F
@Step @RT(14)S_Disconnected @F @F @F @F @RT(0) @F
@AcbCont @RT(7)unnamed @F 0

@Trans @RT(7)Trans25 @F @T @T @T @T @T @TL(2)
sv_bConnect

@RT(7)Trans25 @F

@END_SfcData
@SaActions 0
@SaTrans 0
@SaExits 2
@SaExit @SaText @RT(17)TDisconnectClient 1 @TL(7)
(S_Init.X = FALSE)
AND (S_ReadVersionInfo.X = FALSE)
AND (S_TCPInit.X = FALSE)
AND (S_Disconnecting.X = FALSE)
AND (S_Disconnected.X = FALSE)
AND (sv_bConnect = FALSE)

@RT(15)S_Disconnecting @RT(1)1 @F @F @SaSfc @RT(17)TDisconnectClient 5 @RT(5)DUMMY
@BEG_SfcData 2
@ExitSeq @RT(4)sseq @F 3
@Step @RT(5)Step6 @F @T @F @F @RT(0) @F
@AcbCont @RT(7)unnamed @F 1
@Acb @RT(7)Action8 @F @F @RT(1)N @RT(0) @F @F @T @F

@Trans @RT(6)Trans9 @F @T @T @F @T @T @TL(2)
(*inl.*)

@RT(6)Trans9 @F
@Goto @RT(9)unlabeled @F @F
@END_SfcData

@SaExit @SaText @RT(17)TDisconnectServer 1 @TL(2)
iRequestState = cREQSTATE_SERVICE_CLOSE

@RT(15)S_Disconnecting @RT(1)1 @F @F @SaSfc @RT(17)TDisconnectServer 5 @RT(5)DUMMY
@BEG_SfcData 2
@ExitSeq @RT(4)sseq @F 3
@Step @RT(5)Step6 @F @T @F @F @RT(0) @F
@AcbCont @RT(7)unnamed @F 1
@Acb @RT(7)Action8 @F @F @RT(1)N @RT(0) @F @F @T @F

@Trans @RT(6)Trans9 @F @T @T @F @T @T @TL(2)
(*inl.*)

@RT(6)Trans9 @F
@Goto @RT(9)unlabeled @F @F
@END_SfcData

@END_SfcBody

@@@BEG_Comment@@@
@TL(21)
@h    ! WARNING !
@h    The Kemro K2 system (including software) only meets category B according to EN 954-1,
@h    thus it is not intended for usage in safety-relevant control applications in the field
@h    of personal safety (e.g. emergency stop).
@h    To implement potentially necessary safety-relevant control tasks, always use additional
@h    external safety devices that are intended for the particular purpose, and meet the necessary
@h    functional safety.
@h    For further information see EN 954-1 (EN ISO 13849-1) and/or the K2-x00 user manual, chapter
@h    "CE conformity, directives and standards".

state machine algorithm
when user requests a connection to ServiceNet this algorithm establishes a TCP connection
and sends a client connection message to ServiceNet.
ServiceNet responds by sending a message containing a protocol version information and a "
request state" number which is used to activate this state.
ABParser is used to parse the recieved messages, it provides access to the recieved data via
function aGetXXXValue().
ServiceNet is expected to send a message at least all 30s, otherwise the connection will be closed.
In case of any error (parsing error, timeout, tcp error, ...) the state changes to "Disconnected"
and the algorithm is stopped.

@@@END_Comment@@@
@END_Body

@END_Contents
